C07259=1050.815,63.161,-79.530,170.792,33.398,156.273
C07260=1050.821,63.411,-79.547,170.794,33.400,156.273
C07261=1050.828,63.661,-79.565,170.795,33.402,156.273
C07262=1050.834,63.909,-79.583,170.797,33.404,156.274
C07263=1050.840,64.158,-79.601,170.799,33.406,156.274
C07264=1050.846,64.408,-79.619,170.800,33.407,156.274
C07265=1050.853,64.657,-79.636,170.802,33.410,156.275
C07266=1050.859,64.907,-79.654,170.804,33.412,156.275
C07267=1050.864,65.156,-79.671,170.805,33.414,156.276
C07268=1050.871,65.405,-79.689,170.807,33.416,156.276
C07269=1050.877,65.655,-79.707,170.809,33.418,156.276
C07270=1050.883,65.903,-79.725,170.810,33.420,156.276
C07271=1050.890,66.153,-79.742,170.812,33.422,156.277
C07272=1050.896,66.402,-79.760,170.813,33.424,156.277
C07273=1050.902,66.652,-79.778,170.815,33.426,156.277
C07274=1050.908,66.901,-79.795,170.817,33.428,156.278
C07275=1050.915,67.151,-79.813,170.818,33.430,156.278
C07276=1050.920,67.399,-79.831,170.820,33.432,156.278
C07277=1050.926,67.649,-79.849,170.822,33.434,156.279
C07278=1050.933,67.898,-79.867,170.823,33.436,156.279
C07279=1050.939,68.147,-79.884,170.825,33.438,156.279
C07280=1050.945,68.396,-79.903,170.826,33.440,156.280
C07281=1050.951,68.646,-79.921,170.828,33.442,156.280
C07282=1050.958,68.895,-79.938,170.830,33.444,156.280
C07283=1050.964,69.145,-79.956,170.831,33.446,156.281
C07284=1050.970,69.394,-79.974,170.833,33.449,156.281
C07285=1050.976,69.643,-79.992,170.835,33.451,156.281
C07286=1050.982,69.893,-80.010,170.836,33.453,156.282
C07287=1050.989,70.142,-80.027,170.838,33.455,156.282
C07288=1050.995,70.390,-80.045,170.839,33.457,156.282
C07289=1051.001,70.640,-80.063,170.841,33.459,156.283
C07290=1051.007,70.890,-80.081,170.843,33.461,156.283
C07291=1051.013,71.138,-80.099,170.844,33.463,156.283
C07292=1051.019,71.388,-80.117,170.846,33.465,156.284
C07293=1051.025,71.638,-80.135,170.847,33.467,156.284
C07294=1051.031,71.887,-80.154,170.849,33.469,156.284
C07295=1051.037,72.136,-80.172,170.851,33.471,156.285
C07296=1051.044,72.385,-80.190,170.852,33.473,156.285
C07297=1051.050,72.635,-80.208,170.854,33.475,156.285
C07298=1051.056,72.884,-80.225,170.856,33.478,156.286
C07299=1051.062,73.133,-80.244,170.857,33.479,156.286
C07300=1051.068,73.382,-80.262,170.859,33.481,156.286
C07301=1051.075,73.632,-80.280,170.861,33.483,156.287
C07302=1051.080,73.881,-80.298,170.863,33.485,156.287
C07303=1051.086,74.130,-80.316,170.865,33.487,156.287
C07304=1051.093,74.379,-80.335,170.866,33.490,156.288
C07305=1051.099,74.629,-80.352,170.868,33.492,156.288
C07306=1051.105,74.878,-80.371,170.870,33.494,156.288
C07307=1051.111,75.127,-80.389,170.871,33.496,156.289
C07308=1051.117,75.376,-80.407,170.873,33.498,156.289
C07309=1051.124,75.626,-80.425,170.874,33.500,156.289
C07310=1051.130,75.874,-80.443,170.876,33.502,156.290
C07311=1051.136,76.124,-80.461,170.878,33.504,156.290
C07312=1051.142,76.373,-80.480,170.879,33.506,156.291
C07313=1051.148,76.623,-80.497,170.881,33.508,156.291
C07314=1051.154,76.871,-80.516,170.883,33.510,156.291
C07315=1051.160,77.121,-80.534,170.884,33.512,156.291
C07316=1051.167,77.407,-80.555,170.886,33.515,156.292
C07317=1051.175,77.693,-80.576,170.888,33.517,156.292
C07318=1051.182,77.978,-80.597,170.890,33.519,156.293
C07319=1051.189,78.264,-80.618,170.892,33.522,156.293
C07320=1051.195,78.513,-80.636,170.893,33.524,156.293
C07321=1051.201,78.762,-80.654,170.895,33.526,156.294
C07322=1051.207,79.011,-80.673,170.897,33.528,156.294
C07323=1051.213,79.261,-80.691,170.898,33.530,156.294
C07324=1051.219,79.510,-80.710,170.900,33.532,156.295
C07325=1051.225,79.759,-80.729,170.901,33.534,156.295
C07326=1051.231,80.009,-80.746,170.903,33.536,156.295
C07327=1051.237,80.257,-80.765,170.905,33.538,156.296
C07328=1051.244,80.506,-80.783,170.906,33.541,156.296
C07329=1051.250,80.756,-80.801,170.908,33.543,156.297
C07330=1051.255,81.006,-80.821,170.909,33.545,156.297
C07331=1051.262,81.255,-80.839,170.911,33.547,156.297
C07332=1051.267,81.504,-80.857,170.913,33.549,156.298
C07333=1051.274,81.753,-80.875,170.914,33.551,156.298
C07334=1051.280,82.002,-80.894,170.916,33.553,156.298
C07335=1051.286,82.252,-80.913,170.918,33.555,156.299
C07336=1051.292,82.501,-80.931,170.919,33.558,156.299
C07337=1051.298,82.750,-80.950,170.921,33.560,156.299
C07338=1051.304,82.999,-80.968,170.922,33.562,156.300
C07339=1051.310,83.249,-80.986,170.924,33.564,156.300
C07340=1051.316,83.498,-81.005,170.926,33.566,156.300
C07341=1051.322,83.747,-81.024,170.927,33.568,156.301
C07342=1051.329,83.996,-81.043,170.929,33.570,156.301
C07343=1051.335,84.246,-81.061,170.931,33.572,156.301
C07344=1051.340,84.495,-81.080,170.933,33.574,156.302
C07345=1051.347,84.744,-81.098,170.935,33.576,156.302
C07346=1051.353,84.993,-81.117,170.936,33.579,156.302
C07347=1051.359,85.242,-81.135,170.938,33.580,156.303
C07348=1051.365,85.492,-81.153,170.940,33.582,156.303
C07349=1051.371,85.741,-81.173,170.941,33.584,156.303
C07350=1051.378,85.990,-81.191,170.943,33.586,156.304
C07351=1051.384,86.239,-81.210,170.945,33.589,156.304
C07352=1051.390,86.489,-81.229,170.946,33.591,156.304
C07353=1051.396,86.738,-81.248,170.948,33.593,156.305
C07354=1051.402,86.987,-81.265,170.949,33.595,156.305
C07355=1051.408,87.236,-81.284,170.951,33.597,156.305
C07356=1051.415,87.485,-81.303,170.953,33.599,156.306
C07357=1051.420,87.735,-81.322,170.954,33.601,156.306
C07358=1051.427,87.984,-81.341,170.956,33.603,156.307
C07359=1051.433,88.233,-81.359,170.958,33.605,156.307
C07360=1051.439,88.482,-81.378,170.959,33.607,156.307
C07361=1051.445,88.732,-81.397,170.961,33.609,156.307
C07362=1051.452,88.981,-81.416,170.963,33.612,156.308
C07363=1051.458,89.230,-81.434,170.964,33.614,156.308
C07364=1051.464,89.480,-81.452,170.966,33.616,156.309
C07365=1051.470,89.729,-81.472,170.968,33.618,156.309
C07366=1051.476,89.978,-81.490,170.969,33.620,156.309
C07367=1051.483,90.227,-81.509,170.971,33.622,156.310
C07368=1051.489,90.476,-81.528,170.972,33.624,156.310
C07369=1051.495,90.726,-81.547,170.974,33.626,156.310
C07370=1051.501,90.975,-81.565,170.976,33.628,156.311
C07371=1051.507,91.224,-81.585,170.977,33.631,156.311
C07372=1051.513,91.473,-81.603,170.979,33.633,156.311
C07373=1051.519,91.723,-81.623,170.981,33.634,156.312
C07374=1051.525,91.972,-81.641,170.982,33.636,156.312
C07375=1051.531,92.221,-81.660,170.984,33.639,156.312
C07376=1051.537,92.469,-81.679,170.985,33.641,156.313
C07377=1051.543,92.719,-81.699,170.988,33.643,156.313
C07378=1051.549,92.968,-81.717,170.990,33.645,156.314
C07379=1051.555,93.217,-81.737,170.991,33.647,156.314
C07380=1051.562,93.504,-81.758,170.993,33.650,156.314
C07381=1051.569,93.789,-81.780,170.995,33.652,156.315
C07382=1051.576,94.075,-81.802,170.997,33.655,156.315
C07383=1051.583,94.360,-81.824,170.999,33.657,156.315
C07384=1051.589,94.609,-81.842,171.000,33.659,156.316
C07385=1051.595,94.858,-81.862,171.002,33.662,156.316
C07386=1051.602,95.107,-81.881,171.004,33.664,156.317
C07387=1051.608,95.356,-81.900,171.005,33.666,156.317
C07388=1051.613,95.606,-81.920,171.007,33.667,156.317
C07389=1051.620,95.855,-81.938,171.009,33.670,156.318
C07390=1051.625,96.104,-81.957,171.010,33.672,156.318
C07391=1051.632,96.353,-81.976,171.012,33.674,156.318
C07392=1051.638,96.602,-81.996,171.014,33.676,156.319
C07393=1051.644,96.851,-82.015,171.015,33.678,156.319
C07394=1051.650,97.101,-82.034,171.017,33.680,156.319
C07395=1051.656,97.350,-82.053,171.019,33.682,156.320
C07396=1051.662,97.599,-82.072,171.020,33.684,156.320
C07397=1051.669,97.848,-82.091,171.022,33.687,156.320
C07398=1051.674,98.097,-82.110,171.024,33.689,156.321
C07399=1051.680,98.347,-82.130,171.025,33.691,156.321
C07400=1051.687,98.597,-82.149,171.027,33.693,156.321
C07401=1051.693,98.845,-82.169,171.028,33.695,156.322
C07402=1051.700,99.094,-82.187,171.030,33.697,156.322
C07403=1051.705,99.344,-82.207,171.032,33.699,156.323
C07404=1051.712,99.592,-82.226,171.033,33.701,156.323
C07405=1051.718,99.842,-82.245,171.036,33.704,156.323
C07406=1051.724,100.091,-82.264,171.038,33.706,156.324
C07407=1051.730,100.340,-82.283,171.039,33.708,156.324
C07408=1051.736,100.589,-82.303,171.041,33.710,156.324
C07409=1051.742,100.838,-82.322,171.043,33.712,156.325
C07410=1051.748,101.088,-82.341,171.044,33.714,156.325
C07411=1051.754,101.337,-82.361,171.046,33.716,156.325
C07412=1051.760,101.587,-82.380,171.048,33.719,156.326
C07413=1051.767,101.835,-82.400,171.049,33.721,156.326
C07414=1051.773,102.085,-82.419,171.051,33.723,156.326
C07415=1051.778,102.334,-82.438,171.053,33.725,156.327
C07416=1051.784,102.583,-82.458,171.054,33.727,156.327
C07417=1051.790,102.832,-82.478,171.056,33.729,156.328
C07418=1051.797,103.081,-82.497,171.058,33.732,156.328
C07419=1051.802,103.330,-82.516,171.059,33.733,156.328
C07420=1051.808,103.579,-82.536,171.061,33.735,156.329
C07421=1051.814,103.829,-82.555,171.062,33.738,156.329
C07422=1051.821,104.078,-82.576,171.064,33.740,156.329
C07423=1051.826,104.327,-82.595,171.066,33.742,156.330
C07424=1051.833,104.576,-82.614,171.067,33.744,156.330
C07425=1051.839,104.825,-82.633,171.069,33.746,156.330
C07426=1051.845,105.074,-82.653,171.071,33.748,156.331
C07427=1051.850,105.324,-82.673,171.072,33.751,156.331
C07428=1051.856,105.572,-82.693,171.074,33.753,156.332
C07429=1051.863,105.822,-82.711,171.076,33.755,156.332
C07430=1051.869,106.071,-82.732,171.078,33.757,156.332
C07431=1051.875,106.321,-82.751,171.080,33.759,156.333
C07432=1051.881,106.569,-82.771,171.082,33.761,156.333
C07433=1051.887,106.819,-82.790,171.083,33.764,156.333
C07434=1051.893,107.068,-82.810,171.085,33.766,156.334
C07435=1051.899,107.317,-82.829,171.087,33.768,156.334
C07436=1051.906,107.566,-82.849,171.088,33.770,156.335
C07437=1051.912,107.815,-82.869,171.090,33.772,156.335
C07438=1051.918,108.064,-82.888,171.092,33.774,156.335
C07439=1051.924,108.313,-82.908,171.093,33.777,156.336
C07440=1051.929,108.563,-82.927,171.095,33.779,156.336
C07441=1051.936,108.812,-82.948,171.097,33.781,156.336
C07442=1051.943,109.061,-82.967,171.098,33.783,156.337
C07443=1051.948,109.310,-82.986,171.100,33.785,156.337
C07444=1051.955,109.596,-83.009,171.102,33.788,156.337
C07445=1051.963,109.881,-83.032,171.104,33.790,156.338
C07446=1051.970,110.166,-83.054,171.106,33.792,156.338
C07447=1051.976,110.452,-83.077,171.108,33.795,156.339
C07448=1051.982,110.701,-83.097,171.110,33.797,156.339
C07449=1051.988,110.951,-83.117,171.111,33.799,156.339
C07450=1051.994,111.200,-83.137,171.113,33.801,156.340
C07451=1052.000,111.449,-83.157,171.115,33.803,156.340
C07452=1052.006,111.698,-83.176,171.117,33.806,156.341
C07453=1052.012,111.947,-83.196,171.119,33.808,156.341
C07454=1052.019,112.197,-83.216,171.121,33.810,156.341
C07455=1052.025,112.445,-83.236,171.122,33.812,156.342
C07456=1052.030,112.695,-83.255,171.124,33.814,156.342
C07457=1052.036,112.944,-83.275,171.126,33.816,156.342
C07458=1052.043,113.193,-83.296,171.127,33.819,156.343
C07459=1052.049,113.442,-83.316,171.129,33.821,156.343
C07460=1052.055,113.691,-83.335,171.131,33.823,156.343
C07461=1052.061,113.940,-83.355,171.132,33.825,156.344
C07462=1052.067,114.190,-83.375,171.134,33.827,156.344
C07463=1052.073,114.439,-83.395,171.136,33.830,156.345
C07464=1052.079,114.688,-83.416,171.137,33.831,156.345
C07465=1052.085,114.936,-83.436,171.139,33.834,156.345
C07466=1052.091,115.186,-83.456,171.141,33.836,156.346
C07467=1052.097,115.435,-83.475,171.142,33.838,156.346
C07468=1052.102,115.685,-83.496,171.144,33.840,156.346
C07469=1052.108,115.933,-83.516,171.146,33.843,156.347
C07470=1052.115,116.183,-83.536,171.147,33.845,156.347
C07471=1052.121,116.432,-83.556,171.149,33.847,156.348
C07472=1052.126,116.681,-83.577,171.152,33.849,156.348
C07473=1052.132,116.930,-83.597,171.154,33.852,156.348
C07474=1052.139,117.179,-83.617,171.155,33.854,156.349
C07475=1052.144,117.428,-83.637,171.157,33.856,156.349
C07476=1052.150,117.677,-83.657,171.159,33.858,156.349
C07477=1052.156,117.926,-83.677,171.160,33.860,156.350
C07478=1052.162,118.175,-83.698,171.162,33.863,156.350
C07479=1052.168,118.424,-83.718,171.164,33.865,156.351
C07480=1052.174,118.673,-83.738,171.165,33.867,156.351
C07481=1052.180,118.923,-83.759,171.167,33.869,156.351
C07482=1052.186,119.172,-83.779,171.169,33.872,156.352
C07483=1052.191,119.421,-83.799,171.170,33.874,156.352
C07484=1052.197,119.670,-83.819,171.172,33.876,156.352
C07485=1052.204,119.919,-83.839,171.174,33.878,156.353
C07486=1052.210,120.168,-83.859,171.176,33.880,156.353
C07487=1052.215,120.417,-83.880,171.177,33.883,156.354
C07488=1052.222,120.667,-83.900,171.179,33.885,156.354
C07489=1052.228,120.915,-83.920,171.181,33.887,156.354
C07490=1052.233,121.165,-83.941,171.182,33.889,156.355
C07491=1052.240,121.414,-83.961,171.185,33.892,156.355
C07492=1052.246,121.663,-83.981,171.187,33.894,156.356
C07493=1052.252,121.912,-84.003,171.188,33.896,156.356
C07494=1052.258,122.161,-84.023,171.190,33.898,156.356
C07495=1052.264,122.410,-84.043,171.192,33.900,156.357
C07496=1052.270,122.659,-84.063,171.194,33.903,156.357
C07497=1052.276,122.908,-84.083,171.195,33.905,156.357
C07498=1052.282,123.157,-84.103,171.197,33.907,156.358
C07499=1052.288,123.407,-84.124,171.199,33.909,156.358
C07500=1052.294,123.656,-84.144,171.200,33.911,156.358
C07501=1052.300,123.905,-84.165,171.202,33.914,156.359
C07502=1052.306,124.153,-84.185,171.204,33.916,156.359
C07503=1052.312,124.403,-84.206,171.206,33.918,156.360
C07504=1052.318,124.652,-84.226,171.207,33.920,156.360
C07505=1052.324,124.901,-84.246,171.209,33.922,156.360
C07506=1052.330,125.150,-84.268,171.211,33.925,156.361
C07507=1052.336,125.399,-84.288,171.213,33.926,156.361
C07508=1052.343,125.684,-84.311,171.215,33.929,156.362
C07509=1052.350,125.970,-84.334,171.218,33.932,156.362
C07510=1052.357,126.256,-84.358,171.220,33.934,156.362
C07511=1052.364,126.541,-84.382,171.222,33.937,156.363
C07512=1052.370,126.790,-84.402,171.223,33.939,156.363
C07513=1052.377,127.039,-84.423,171.225,33.941,156.364
C07514=1052.382,127.288,-84.443,171.227,33.943,156.364
C07515=1052.389,127.537,-84.463,171.229,33.945,156.364
C07516=1052.394,127.786,-84.485,171.230,33.948,156.365
C07517=1052.401,128.036,-84.505,171.232,33.950,156.365
C07518=1052.407,128.284,-84.525,171.234,33.952,156.366
C07519=1052.413,128.534,-84.546,171.236,33.954,156.366
C07520=1052.419,128.782,-84.567,171.237,33.956,156.366
C07521=1052.426,129.032,-84.587,171.239,33.958,156.367
C07522=1052.431,129.281,-84.608,171.241,33.960,156.367
C07523=1052.438,129.530,-84.629,171.243,33.963,156.367
C07524=1052.444,129.779,-84.648,171.244,33.965,156.368
C07525=1052.450,130.028,-84.670,171.246,33.967,156.368
C07526=1052.456,130.277,-84.690,171.249,33.969,156.369
C07527=1052.462,130.527,-84.711,171.251,33.971,156.369
C07528=1052.468,130.775,-84.732,171.252,33.973,156.369
C07529=1052.475,131.024,-84.752,171.254,33.976,156.370
C07530=1052.481,131.273,-84.774,171.256,33.978,156.370
C07531=1052.487,131.522,-84.794,171.258,33.980,156.370
C07532=1052.493,131.772,-84.815,171.259,33.982,156.371
C07533=1052.499,132.020,-84.835,171.261,33.985,156.371
C07534=1052.505,132.270,-84.856,171.263,33.987,156.371
C07535=1052.511,132.519,-84.877,171.265,33.989,156.372
C07536=1052.517,132.768,-84.898,171.266,33.991,156.372
C07537=1052.523,133.017,-84.919,171.268,33.994,156.373
C07538=1052.529,133.266,-84.940,171.270,33.996,156.373
C07539=1052.535,133.515,-84.961,171.272,33.998,156.373
C07540=1052.541,133.764,-84.982,171.273,34.000,156.374
C07541=1052.546,134.013,-85.003,171.275,34.003,156.374
C07542=1052.553,134.262,-85.024,171.278,34.005,156.375
C07543=1052.559,134.511,-85.044,171.280,34.007,156.375
C07544=1052.565,134.760,-85.066,171.282,34.009,156.375
C07545=1052.571,135.009,-85.086,171.283,34.012,156.376
C07546=1052.577,135.258,-85.108,171.285,34.014,156.376
C07547=1052.582,135.507,-85.129,171.287,34.016,156.377
C07548=1052.589,135.756,-85.149,171.289,34.018,156.377
C07549=1052.595,136.005,-85.171,171.290,34.021,156.377
C07550=1052.600,136.255,-85.191,171.292,34.022,156.378
C07551=1052.607,136.503,-85.212,171.294,34.025,156.378
C07552=1052.613,136.752,-85.234,171.296,34.027,156.378
C07553=1052.619,137.002,-85.255,171.298,34.030,156.379
C07554=1052.625,137.250,-85.275,171.299,34.031,156.379
C07555=1052.631,137.499,-85.297,171.301,34.034,156.380
C07556=1052.637,137.749,-85.318,171.303,34.036,156.380
C07557=1052.643,137.998,-85.339,171.306,34.038,156.380
C07558=1052.650,138.246,-85.360,171.307,34.041,156.381
C07559=1052.655,138.496,-85.381,171.309,34.043,156.381
C07560=1052.661,138.745,-85.402,171.311,34.045,156.382
C07561=1052.667,138.994,-85.424,171.313,34.047,156.382
C07562=1052.673,139.242,-85.445,171.315,34.050,156.382
C07563=1052.679,139.492,-85.466,171.316,34.052,156.383
C07564=1052.685,139.741,-85.487,171.318,34.054,156.383
C07565=1052.691,139.990,-85.508,171.320,34.056,156.384
C07566=1052.697,140.239,-85.530,171.322,34.059,156.384
C07567=1052.702,140.488,-85.551,171.324,34.061,156.384
C07568=1052.709,140.737,-85.572,171.325,34.063,156.385
C07569=1052.715,140.986,-85.593,171.327,34.066,156.385
C07570=1052.721,141.235,-85.615,171.329,34.068,156.386
C07571=1052.727,141.484,-85.636,171.332,34.070,156.386
C07572=1052.733,141.770,-85.660,171.334,34.073,156.386
C07573=1052.741,142.054,-85.685,171.336,34.075,156.387
C07574=1052.747,142.339,-85.710,171.338,34.078,156.387
C07575=1052.754,142.625,-85.734,171.340,34.081,156.388
C07576=1052.760,142.874,-85.756,171.342,34.083,156.388
C07577=1052.767,143.123,-85.777,171.344,34.086,156.389
C07578=1052.772,143.372,-85.798,171.345,34.088,156.389
C07579=1052.778,143.621,-85.820,171.347,34.090,156.389
C07580=1052.785,143.870,-85.841,171.349,34.092,156.390
C07581=1052.790,144.119,-85.863,171.351,34.095,156.390
C07582=1052.796,144.368,-85.884,171.353,34.097,156.391
C07583=1052.802,144.617,-85.906,171.355,34.099,156.391
C07584=1052.808,144.866,-85.926,171.357,34.102,156.391
C07585=1052.814,145.115,-85.948,171.359,34.103,156.392
C07586=1052.820,145.365,-85.970,171.361,34.106,156.392
C07587=1052.826,145.614,-85.991,171.363,34.108,156.393
C07588=1052.832,145.862,-86.013,171.365,34.111,156.393
C07589=1052.838,146.111,-86.034,171.367,34.113,156.393
C07590=1052.844,146.361,-86.056,171.368,34.115,156.394
C07591=1052.850,146.609,-86.077,171.370,34.117,156.394
C07592=1052.856,146.858,-86.099,171.372,34.119,156.395
C07593=1052.862,147.108,-86.120,171.374,34.122,156.395
C07594=1052.868,147.357,-86.142,171.376,34.124,156.395
C07595=1052.874,147.605,-86.164,171.378,34.126,156.396
C07596=1052.880,147.854,-86.186,171.379,34.129,156.396
C07597=1052.886,148.103,-86.207,171.381,34.131,156.397
C07598=1052.892,148.352,-86.229,171.384,34.133,156.397
C07599=1052.898,148.601,-86.250,171.386,34.136,156.397
C07600=1052.904,148.850,-86.272,171.388,34.138,156.398
C07601=1052.910,149.099,-86.293,171.390,34.140,156.398
C07602=1052.917,149.348,-86.315,171.391,34.143,156.399
C07603=1052.922,149.597,-86.336,171.393,34.145,156.399
C07604=1052.928,149.846,-86.359,171.395,34.147,156.399
C07605=1052.934,150.095,-86.381,171.397,34.150,156.400
C07606=1052.940,150.344,-86.403,171.399,34.152,156.400
C07607=1052.946,150.593,-86.424,171.401,34.154,156.401
C07608=1052.952,150.842,-86.445,171.403,34.157,156.401
C07609=1052.958,151.090,-86.468,171.404,34.159,156.401
C07610=1052.964,151.340,-86.490,171.407,34.161,156.402
C07611=1052.970,151.589,-86.512,171.409,34.164,156.402
C07612=1052.975,151.838,-86.533,171.411,34.166,156.403
C07613=1052.982,152.086,-86.555,171.413,34.168,156.403
C07614=1052.988,152.336,-86.577,171.415,34.171,156.404
C07615=1052.994,152.585,-86.599,171.417,34.173,156.404
C07616=1053.000,152.834,-86.621,171.418,34.175,156.404
C07617=1053.006,153.082,-86.643,171.420,34.178,156.405
C07618=1053.012,153.331,-86.664,171.422,34.180,156.405
C07619=1053.018,153.581,-86.686,171.424,34.182,156.406
C07620=1053.023,153.830,-86.708,171.426,34.185,156.406
C07621=1053.030,154.079,-86.731,171.428,34.187,156.406
C07622=1053.036,154.328,-86.752,171.431,34.189,156.407
C07623=1053.042,154.576,-86.774,171.433,34.192,156.407
C07624=1053.047,154.825,-86.796,171.434,34.194,156.408
C07625=1053.053,155.074,-86.818,171.436,34.196,156.408
C07626=1053.060,155.323,-86.840,171.438,34.199,156.409
C07627=1053.065,155.573,-86.863,171.440,34.201,156.409
C07628=1053.071,155.822,-86.884,171.442,34.203,156.409
C07629=1053.077,156.070,-86.906,171.444,34.206,156.410
C07630=1053.083,156.319,-86.929,171.446,34.208,156.410
C07631=1053.089,156.568,-86.951,171.448,34.211,156.411
C07632=1053.095,156.817,-86.973,171.450,34.213,156.411
C07633=1053.101,157.066,-86.995,171.451,34.215,156.411
C07634=1053.107,157.315,-87.017,171.454,34.218,156.412
C07635=1053.113,157.564,-87.039,171.456,34.220,156.412
C07636=1053.120,157.849,-87.064,171.458,34.223,156.413
C07637=1053.127,158.134,-87.089,171.461,34.225,156.413
C07638=1053.134,158.418,-87.115,171.463,34.228,156.414
C07639=1053.141,158.704,-87.140,171.465,34.231,156.414
C07640=1053.146,158.952,-87.163,171.467,34.233,156.415
C07641=1053.152,159.201,-87.185,171.469,34.236,156.415
C07642=1053.158,159.450,-87.208,171.471,34.238,156.415
C07643=1053.164,159.700,-87.229,171.473,34.241,156.416
C07644=1053.171,159.948,-87.252,171.475,34.243,156.416
C07645=1053.176,160.198,-87.274,171.477,34.245,156.417
C07646=1053.183,160.446,-87.296,171.479,34.248,156.417
C07647=1053.189,160.695,-87.318,171.481,34.250,156.417
C07648=1053.194,160.944,-87.341,171.483,34.252,156.418
C07649=1053.200,161.193,-87.364,171.485,34.255,156.418
C07650=1053.206,161.443,-87.386,171.487,34.257,156.419
C07651=1053.212,161.691,-87.408,171.489,34.260,156.419
C07652=1053.217,161.940,-87.431,171.491,34.262,156.420
C07653=1053.223,162.189,-87.453,171.493,34.265,156.420
C07654=1053.228,162.438,-87.476,171.495,34.267,156.421
C07655=1053.235,162.687,-87.498,171.498,34.270,156.421
C07656=1053.241,162.935,-87.521,171.499,34.272,156.422
C07657=1053.246,163.185,-87.544,171.501,34.275,156.422
C07658=1053.252,163.434,-87.566,171.503,34.277,156.422
C07659=1053.258,163.682,-87.589,171.505,34.280,156.423
C07660=1053.264,163.931,-87.612,171.507,34.282,156.423
C07661=1053.269,164.181,-87.634,171.509,34.285,156.424
C07662=1053.274,164.429,-87.657,171.511,34.287,156.424
C07663=1053.281,164.678,-87.679,171.513,34.289,156.425
C07664=1053.287,164.927,-87.702,171.515,34.292,156.425
C07665=1053.292,165.175,-87.725,171.517,34.294,156.425
C07666=1053.298,165.425,-87.747,171.520,34.297,156.426
C07667=1053.304,165.674,-87.769,171.522,34.299,156.426
C07668=1053.310,165.922,-87.792,171.524,34.302,156.427
C07669=1053.316,166.171,-87.815,171.525,34.304,156.427
C07670=1053.321,166.420,-87.838,171.527,34.307,156.428
C07671=1053.327,166.669,-87.861,171.529,34.309,156.428
C07672=1053.334,166.918,-87.884,171.531,34.312,156.429
C07673=1053.339,167.167,-87.906,171.533,34.315,156.429
C07674=1053.345,167.416,-87.929,171.535,34.317,156.430
C07675=1053.351,167.665,-87.952,171.538,34.320,156.430
C07676=1053.357,167.914,-87.974,171.540,34.322,156.430
C07677=1053.363,168.162,-87.997,171.542,34.324,156.431
C07678=1053.368,168.411,-88.020,171.544,34.327,156.431
C07679=1053.374,168.660,-88.043,171.546,34.329,156.432
C07680=1053.380,168.909,-88.066,171.548,34.332,156.432
C07681=1053.386,169.158,-88.089,171.550,34.334,156.433
C07682=1053.392,169.407,-88.111,171.552,34.337,156.433
C07683=1053.398,169.656,-88.134,171.554,34.339,156.433
C07684=1053.404,169.904,-88.157,171.556,34.342,156.434
C07685=1053.409,170.153,-88.180,171.559,34.344,156.434
C07686=1053.415,170.402,-88.203,171.561,34.347,156.435
C07687=1053.422,170.651,-88.225,171.563,34.349,156.435
C07688=1053.428,170.900,-88.249,171.565,34.352,156.436
C07689=1053.434,171.149,-88.271,171.567,34.354,156.436
C07690=1053.439,171.398,-88.294,171.569,34.357,156.437
C07691=1053.445,171.647,-88.317,171.571,34.359,156.437
C07692=1053.451,171.896,-88.340,171.573,34.362,156.438
C07693=1053.457,172.145,-88.363,171.575,34.364,156.438
C07694=1053.463,172.393,-88.386,171.577,34.366,156.438
C07695=1053.469,172.642,-88.409,171.580,34.369,156.439
C07696=1053.474,172.891,-88.432,171.582,34.371,156.439
C07697=1053.481,173.141,-88.455,171.584,34.374,156.440
C07698=1053.487,173.389,-88.478,171.586,34.376,156.440
C07699=1053.493,173.638,-88.501,171.588,34.379,156.441
C07700=1053.499,173.923,-88.527,171.590,34.382,156.441
C07701=1053.507,174.206,-88.554,171.592,34.384,156.442
C07702=1053.513,174.492,-88.580,171.595,34.388,156.442
C07703=1053.520,174.776,-88.606,171.597,34.390,156.443
C07704=1053.526,175.025,-88.629,171.600,34.393,156.443
C07705=1053.532,175.273,-88.652,171.602,34.395,156.444
C07706=1053.538,175.522,-88.675,171.604,34.398,156.444
C07707=1053.544,175.772,-88.699,171.606,34.400,156.444
C07708=1053.550,176.021,-88.722,171.608,34.403,156.445
C07709=1053.557,176.269,-88.745,171.610,34.405,156.445
C07710=1053.562,176.518,-88.768,171.612,34.408,156.446
C07711=1053.568,176.767,-88.791,171.614,34.410,156.446
C07712=1053.574,177.016,-88.814,171.616,34.413,156.447
C07713=1053.580,177.264,-88.838,171.620,34.415,156.447
C07714=1053.586,177.513,-88.861,171.622,34.418,156.448
C07715=1053.592,177.762,-88.883,171.624,34.420,156.448
C07716=1053.599,178.011,-88.907,171.626,34.423,156.449
C07717=1053.605,178.260,-88.930,171.628,34.425,156.449
C07718=1053.611,178.509,-88.953,171.630,34.427,156.449
C07719=1053.617,178.757,-88.976,171.632,34.430,156.450
C07720=1053.623,179.007,-89.000,171.634,34.432,156.450
C07721=1053.629,179.255,-89.023,171.636,34.435,156.451
C07722=1053.635,179.504,-89.046,171.639,34.437,156.451
C07723=1053.641,179.753,-89.069,171.641,34.440,156.452
C07724=1053.647,180.002,-89.093,171.643,34.442,156.452
C07725=1053.653,180.251,-89.116,171.645,34.445,156.453
C07726=1053.659,180.499,-89.139,171.647,34.447,156.453
C07727=1053.665,180.748,-89.163,171.650,34.450,156.453
C07728=1053.672,180.997,-89.186,171.652,34.452,156.454
C07729=1053.678,181.246,-89.209,171.654,34.455,156.454
C07730=1053.684,181.495,-89.233,171.656,34.457,156.455
C07731=1053.690,181.744,-89.256,171.659,34.460,156.455
C07732=1053.696,181.992,-89.279,171.661,34.462,156.456
C07733=1053.702,182.242,-89.303,171.663,34.465,156.456
C07734=1053.708,182.490,-89.326,171.665,34.468,156.457
C07735=1053.714,182.739,-89.349,171.667,34.470,156.457
C07736=1053.721,182.988,-89.373,171.669,34.473,156.458
C07737=1053.726,183.237,-89.396,171.672,34.475,156.458
C07738=1053.733,183.486,-89.420,171.674,34.478,156.458
C07739=1053.739,183.735,-89.443,171.677,34.480,156.459
C07740=1053.745,183.983,-89.467,171.679,34.483,156.459
C07741=1053.751,184.232,-89.490,171.681,34.485,156.460
C07742=1053.757,184.481,-89.514,171.683,34.488,156.460
C07743=1053.762,184.729,-89.538,171.685,34.490,156.461
C07744=1053.769,184.979,-89.561,171.687,34.493,156.461
C07745=1053.775,185.227,-89.585,171.689,34.496,156.462
C07746=1053.780,185.476,-89.609,171.691,34.498,156.462
C07747=1053.786,185.725,-89.632,171.695,34.501,156.463
C07748=1053.792,185.974,-89.657,171.697,34.504,156.463
C07749=1053.798,186.222,-89.680,171.699,34.506,156.464
C07750=1053.803,186.471,-89.705,171.701,34.509,156.464
C07751=1053.809,186.720,-89.728,171.703,34.512,156.465
C07752=1053.815,186.969,-89.752,171.705,34.514,156.465
C07753=1053.821,187.217,-89.776,171.707,34.517,156.466
C07754=1053.827,187.466,-89.800,171.709,34.519,156.466
C07755=1053.832,187.715,-89.823,171.712,34.523,156.467
C07756=1053.838,187.964,-89.847,171.715,34.525,156.467
C07757=1053.844,188.213,-89.872,171.717,34.528,156.468
C07758=1053.850,188.461,-89.895,171.719,34.531,156.468
C07759=1053.856,188.710,-89.920,171.721,34.533,156.469
C07760=1053.862,188.959,-89.943,171.723,34.536,156.469
C07761=1053.867,189.208,-89.967,171.725,34.538,156.470
C07762=1053.873,189.456,-89.991,171.728,34.541,156.470
C07763=1053.879,189.706,-90.016,171.730,34.544,156.471
C07764=1053.886,189.990,-90.043,171.733,34.547,156.471
C07765=1053.892,190.273,-90.070,171.735,34.550,156.472
C07766=1053.900,190.558,-90.098,171.738,34.553,156.472
C07767=1053.906,190.842,-90.125,171.740,34.556,156.473
C07768=1053.912,191.090,-90.149,171.742,34.559,156.473
C07769=1053.918,191.339,-90.174,171.746,34.561,156.474
C07770=1053.924,191.587,-90.197,171.748,34.564,156.474
C07771=1053.930,191.837,-90.221,171.750,34.567,156.475
C07772=1053.936,192.086,-90.245,171.752,34.569,156.475
C07773=1053.942,192.335,-90.269,171.754,34.573,156.476
C07774=1053.948,192.583,-90.293,171.756,34.575,156.476
C07775=1053.954,192.833,-90.318,171.759,34.578,156.477
C07776=1053.960,193.081,-90.341,171.761,34.581,156.477
C07777=1053.966,193.330,-90.366,171.764,34.583,156.478
C07778=1053.972,193.578,-90.390,171.766,34.586,156.478
C07779=1053.978,193.827,-90.415,171.768,34.589,156.479
C07780=1053.984,194.075,-90.439,171.770,34.591,156.479
C07781=1053.990,194.325,-90.463,171.773,34.594,156.480
C07782=1053.996,194.573,-90.487,171.775,34.597,156.480
C07783=1054.002,194.822,-90.512,171.777,34.599,156.481
C07784=1054.007,195.071,-90.536,171.780,34.602,156.481
C07785=1054.014,195.320,-90.560,171.782,34.605,156.482
C07786=1054.019,195.568,-90.584,171.785,34.608,156.482
C07787=1054.026,195.817,-90.608,171.787,34.610,156.483
C07788=1054.031,196.066,-90.632,171.789,34.613,156.483
C07789=1054.038,196.314,-90.657,171.791,34.616,156.484
C07790=1054.043,196.563,-90.681,171.793,34.618,156.484
C07791=1054.050,196.812,-90.705,171.797,34.621,156.485
C07792=1054.056,197.061,-90.730,171.799,34.624,156.485
C07793=1054.062,197.309,-90.754,171.801,34.627,156.486
C07794=1054.068,197.559,-90.778,171.803,34.629,156.486
C07795=1054.073,197.807,-90.803,171.806,34.632,156.487
C07796=1054.080,198.056,-90.827,171.808,34.635,156.487
C07797=1054.085,198.304,-90.852,171.810,34.637,156.488
C07798=1054.092,198.553,-90.876,171.813,34.640,156.488
C07799=1054.098,198.802,-90.901,171.815,34.643,156.489
C07800=1054.104,199.050,-90.925,171.818,34.646,156.489
C07801=1054.110,199.299,-90.949,171.820,34.649,156.490
C07802=1054.116,199.549,-90.974,171.822,34.651,156.490
C07803=1054.122,199.796,-90.998,171.824,34.654,156.491
C07804=1054.128,200.046,-91.023,171.827,34.657,156.491
C07805=1054.135,200.295,-91.047,171.830,34.659,156.492
C07806=1054.140,200.543,-91.072,171.832,34.662,156.492
C07807=1054.147,200.792,-91.096,171.835,34.665,156.493
C07808=1054.153,201.041,-91.120,171.837,34.667,156.493
C07809=1054.159,201.289,-91.145,171.839,34.670,156.494
C07810=1054.165,201.538,-91.169,171.841,34.673,156.494
C07811=1054.171,201.786,-91.195,171.845,34.676,156.495
C07812=1054.177,202.035,-91.219,171.847,34.678,156.495
C07813=1054.183,202.284,-91.244,171.849,34.682,156.496
C07814=1054.189,202.533,-91.268,171.851,34.684,156.496
C07815=1054.195,202.781,-91.293,171.854,34.687,156.497
C07816=1054.201,203.030,-91.318,171.856,34.690,156.498
C07817=1054.206,203.279,-91.342,171.858,34.693,156.498
C07818=1054.213,203.527,-91.368,171.861,34.696,156.499
C07819=1054.218,203.777,-91.392,171.864,34.698,156.499
C07820=1054.224,204.024,-91.417,171.866,34.701,156.500
C07821=1054.230,204.273,-91.443,171.868,34.705,156.500
C07822=1054.236,204.522,-91.467,171.870,34.707,156.501
C07823=1054.242,204.771,-91.493,171.873,34.710,156.501
C07824=1054.248,205.019,-91.516,171.876,34.713,156.502
C07825=1054.255,205.268,-91.542,171.878,34.716,156.502
C07826=1054.260,205.517,-91.566,171.881,34.719,156.503
C07827=1054.266,205.765,-91.591,171.883,34.721,156.503
C07828=1054.291,206.816,-91.697,172.092,34.813,156.518
C07829=1054.298,207.059,-91.722,172.094,34.817,156.519
C07830=1054.304,207.301,-91.748,172.096,34.821,156.520
C07831=1054.311,207.543,-91.772,172.098,34.824,156.520
C07832=1054.316,207.785,-91.797,172.100,34.828,156.521
C07833=1054.323,208.027,-91.823,172.101,34.832,156.522
C07834=1054.329,208.269,-91.848,172.104,34.835,156.523
C07835=1054.335,208.511,-91.873,172.106,34.839,156.523
C07836=1054.341,208.753,-91.898,172.107,34.842,156.524
C07837=1054.347,209.001,-91.924,172.109,34.846,156.525
C07838=1054.353,209.251,-91.951,172.112,34.850,156.525
C07839=1054.360,209.499,-91.977,172.114,34.853,156.526
C07840=1054.366,209.748,-92.002,172.115,34.857,156.527
C07841=1054.373,209.996,-92.028,172.117,34.861,156.528
C07842=1054.379,210.245,-92.055,172.120,34.864,156.528
C07843=1054.385,210.493,-92.081,172.122,34.868,156.529
C07844=1054.392,210.741,-92.107,172.123,34.872,156.530
C07845=1054.397,210.990,-92.133,172.125,34.876,156.530
C07846=1054.404,211.239,-92.159,172.128,34.879,156.531
C07847=1054.410,211.488,-92.186,172.130,34.883,156.532
C07848=1054.416,211.736,-92.211,172.131,34.886,156.533
C07849=1054.423,211.984,-92.237,172.133,34.890,156.533
C07850=1054.429,212.233,-92.264,172.136,34.894,156.534
C07851=1054.436,212.481,-92.290,172.138,34.897,156.535
C07852=1054.441,212.730,-92.316,172.139,34.901,156.535
C07853=1054.448,212.979,-92.342,172.141,34.905,156.536
C07854=1054.454,213.227,-92.369,172.143,34.908,156.537
C07855=1054.460,213.475,-92.395,172.146,34.912,156.538
C07856=1054.466,213.724,-92.421,172.147,34.916,156.538
C07857=1054.473,213.973,-92.447,172.149,34.920,156.539
C07858=1054.479,214.222,-92.474,172.152,34.923,156.540
C07859=1054.485,214.470,-92.500,172.154,34.927,156.541
C07860=1054.492,214.719,-92.527,172.155,34.930,156.541
C07861=1054.498,214.967,-92.553,172.157,34.934,156.542
C07862=1054.504,215.216,-92.579,172.160,34.938,156.543
C07863=1054.510,215.464,-92.605,172.162,34.941,156.543
C07864=1054.517,215.713,-92.632,172.164,34.945,156.544
C07865=1054.523,215.961,-92.658,172.165,34.949,156.545
C07866=1054.529,216.210,-92.685,172.168,34.952,156.546
C07867=1054.535,216.458,-92.712,172.170,34.956,156.546
C07868=1054.542,216.706,-92.738,172.172,34.959,156.547
C07869=1054.548,216.956,-92.764,172.174,34.963,156.548
C07870=1054.554,217.204,-92.790,172.176,34.967,156.549
C07871=1054.560,217.452,-92.817,172.178,34.971,156.549
C07872=1054.567,217.701,-92.843,172.180,34.975,156.550
C07873=1054.573,217.950,-92.870,172.182,34.978,156.551
C07874=1054.580,218.198,-92.897,172.185,34.982,156.551
C07875=1054.586,218.447,-92.923,172.186,34.985,156.552
C07876=1054.592,218.695,-92.950,172.188,34.989,156.553
C07877=1054.599,218.944,-92.976,172.190,34.993,156.554
C07878=1054.605,219.192,-93.003,172.193,34.996,156.554
C07879=1054.612,219.441,-93.029,172.195,34.999,156.555
C07880=1054.617,219.689,-93.056,172.197,35.003,156.556
C07881=1054.623,219.938,-93.083,172.198,35.006,156.556
C07882=1054.630,220.186,-93.109,172.201,35.010,156.557
C07883=1054.636,220.435,-93.136,172.203,35.014,156.558
C07884=1054.643,220.683,-93.162,172.205,35.017,156.559
C07885=1054.649,220.927,-93.189,172.207,35.021,156.559
C07886=1054.655,221.173,-93.215,172.210,35.025,156.560
C07887=1054.662,221.417,-93.241,172.211,35.028,156.561
C07888=1054.667,221.662,-93.268,172.213,35.032,156.561
C07889=1054.674,221.906,-93.294,172.215,35.035,156.562
C07890=1054.680,222.151,-93.321,172.218,35.039,156.563
C07891=1054.686,222.396,-93.347,172.220,35.043,156.564
C07892=1054.692,222.641,-93.374,172.222,35.046,156.564
C07893=1054.699,222.888,-93.400,172.223,35.050,156.565
C07894=1054.705,223.137,-93.427,172.226,35.053,156.566
C07895=1054.711,223.386,-93.454,172.228,35.057,156.566
C07896=1054.717,223.635,-93.481,172.230,35.061,156.567
C07897=1054.723,223.883,-93.508,172.233,35.064,156.568
C07898=1054.730,224.132,-93.536,172.235,35.068,156.569
C07899=1054.736,224.380,-93.562,172.237,35.072,156.569
C07900=1054.742,224.628,-93.588,172.238,35.075,156.570
C07901=1054.749,224.877,-93.616,172.241,35.079,156.571
C07902=1054.755,225.126,-93.643,172.243,35.082,156.571
C07903=1054.761,225.374,-93.670,172.245,35.086,156.572
C07904=1054.767,225.622,-93.697,172.247,35.090,156.573
C07905=1054.773,225.871,-93.724,172.250,35.093,156.574
C07906=1054.780,226.120,-93.750,172.252,35.097,156.574
C07907=1054.786,226.367,-93.778,172.254,35.100,156.575
C07908=1054.793,226.616,-93.805,172.256,35.104,156.576
C07909=1054.799,226.865,-93.831,172.259,35.107,156.576
C07910=1054.805,227.113,-93.859,172.260,35.111,156.577
C07911=1054.811,227.361,-93.886,172.262,35.114,156.578
C07912=1054.818,227.610,-93.914,172.264,35.118,156.579
C07913=1054.825,227.859,-93.940,172.267,35.121,156.579
C07914=1054.831,228.106,-93.967,172.269,35.125,156.580
C07915=1054.837,228.355,-93.994,172.271,35.129,156.581
C07916=1054.843,228.604,-94.021,172.274,35.132,156.581
C07917=1054.850,228.852,-94.049,172.276,35.136,156.582
C07918=1054.856,229.101,-94.076,172.278,35.139,156.583
C07919=1054.862,229.349,-94.103,172.280,35.143,156.584
C07920=1054.869,229.598,-94.130,172.283,35.147,156.584
C07921=1054.875,229.846,-94.157,172.285,35.150,156.585
C07922=1054.881,230.095,-94.184,172.287,35.154,156.586
C07923=1054.887,230.343,-94.212,172.289,35.157,156.586
C07924=1054.894,230.591,-94.240,172.291,35.161,156.587
C07925=1054.900,230.840,-94.267,172.293,35.165,156.588
C07926=1054.906,231.088,-94.294,172.295,35.168,156.589
C07927=1054.912,231.337,-94.322,172.298,35.171,156.589
C07928=1054.919,231.586,-94.349,172.300,35.175,156.590
C07929=1054.925,231.833,-94.377,172.302,35.178,156.591
C07930=1054.931,232.083,-94.404,172.304,35.182,156.591
C07931=1054.937,232.330,-94.431,172.307,35.186,156.592
C07932=1054.944,232.579,-94.459,172.309,35.189,156.593
C07933=1054.950,232.828,-94.486,172.311,35.193,156.594
C07934=1054.956,233.076,-94.513,172.314,35.197,156.594
C07935=1054.962,233.324,-94.541,172.316,35.200,156.595
C07936=1054.969,233.573,-94.569,172.318,35.204,156.596
C07937=1054.975,233.821,-94.596,172.320,35.207,156.596
C07938=1054.981,234.070,-94.624,172.323,35.211,156.597
C07939=1054.987,234.318,-94.652,172.325,35.215,156.598
C07940=1054.993,234.566,-94.679,172.327,35.218,156.599
C07941=1055.000,234.807,-94.706,172.330,35.222,156.599
C07942=1055.005,235.048,-94.732,172.332,35.225,156.600
C07943=1055.012,235.289,-94.759,172.334,35.228,156.601
C07944=1055.018,235.530,-94.786,172.335,35.232,156.601
C07945=1055.024,235.770,-94.812,172.338,35.235,156.602
C07946=1055.029,236.011,-94.840,172.340,35.239,156.603
C07947=1055.036,236.252,-94.866,172.342,35.242,156.603
C07948=1055.042,236.493,-94.893,172.344,35.246,156.604
C07949=1055.048,236.741,-94.921,172.347,35.249,156.605
C07950=1055.054,236.989,-94.949,172.349,35.253,156.606
C07951=1055.061,237.238,-94.976,172.351,35.256,156.606
C07952=1055.067,237.486,-95.005,172.354,35.260,156.607
C07953=1055.074,237.735,-95.032,172.356,35.264,156.608
C07954=1055.080,237.982,-95.060,172.358,35.267,156.608
C07955=1055.086,238.231,-95.088,172.360,35.271,156.609
C07956=1055.092,238.480,-95.116,172.363,35.274,156.610
C07957=1055.099,238.729,-95.143,172.365,35.277,156.611
C07958=1055.106,238.977,-95.170,172.367,35.281,156.611
C07959=1055.111,239.225,-95.198,172.370,35.285,156.612
C07960=1055.118,239.473,-95.227,172.372,35.288,156.613
C07961=1055.125,239.721,-95.255,172.375,35.292,156.613
C07962=1055.130,239.970,-95.283,172.377,35.295,156.614
C07963=1055.137,240.218,-95.310,172.380,35.299,156.615
C07964=1055.143,240.466,-95.338,172.382,35.303,156.616
C07965=1055.149,240.715,-95.366,172.384,35.306,156.616
C07966=1055.156,240.964,-95.394,172.387,35.310,156.617
C07967=1055.162,241.212,-95.422,172.389,35.313,156.618
C07968=1055.168,241.461,-95.450,172.391,35.316,156.618
C07969=1055.175,241.709,-95.477,172.394,35.320,156.619
C07970=1055.181,241.957,-95.506,172.396,35.324,156.620
C07971=1055.187,242.206,-95.534,172.398,35.327,156.621
C07972=1055.193,242.454,-95.563,172.400,35.331,156.621
C07973=1055.200,242.702,-95.590,172.403,35.334,156.622
C07974=1055.205,242.950,-95.618,172.405,35.338,156.623
C07975=1055.211,243.199,-95.647,172.407,35.341,156.623
C07976=1055.218,243.447,-95.675,172.410,35.345,156.624
C07977=1055.224,243.696,-95.703,172.412,35.349,156.625
C07978=1055.231,243.944,-95.731,172.415,35.352,156.626
C07979=1055.237,244.193,-95.759,172.418,35.356,156.626
C07980=1055.243,244.440,-95.787,172.420,35.359,156.627
C07981=1055.249,244.689,-95.816,172.422,35.363,156.628
C07982=1055.255,244.937,-95.844,172.424,35.367,156.629
C07983=1055.262,245.185,-95.873,172.427,35.370,156.629
C07984=1055.268,245.434,-95.901,172.429,35.373,156.630
C07985=1055.275,245.683,-95.929,172.431,35.377,156.631
C07986=1055.281,245.931,-95.958,172.434,35.380,156.631
C07987=1055.287,246.179,-95.986,172.436,35.384,156.632
C07988=1055.293,246.427,-96.013,172.438,35.387,156.633
C07989=1055.299,246.675,-96.042,172.442,35.391,156.634
C07990=1055.305,246.924,-96.071,172.444,35.395,156.634
C07991=1055.312,247.172,-96.100,172.446,35.398,156.635
C07992=1055.318,247.421,-96.128,172.448,35.402,156.636
C07993=1055.324,247.669,-96.157,172.451,35.405,156.636
C07994=1055.330,247.917,-96.185,172.453,35.409,156.637
C07995=1055.336,248.165,-96.214,172.455,35.413,156.638
C07996=1055.342,248.414,-96.242,172.458,35.417,156.639
C07997=1055.348,248.652,-96.269,172.460,35.420,156.639
C07998=1055.354,248.889,-96.297,172.462,35.423,156.640
C07999=1055.360,249.127,-96.325,172.465,35.427,156.641
C08000=1055.366,249.365,-96.352,172.467,35.430,156.642
C08001=1055.371,249.602,-96.379,172.469,35.433,156.642
C08002=1055.377,249.841,-96.406,172.472,35.437,156.643
C08003=1055.384,250.078,-96.434,172.475,35.441,156.644
C08004=1055.390,250.316,-96.461,172.477,35.444,156.644
C08005=1055.396,250.564,-96.490,172.479,35.447,156.645
C08006=1055.402,250.813,-96.519,172.482,35.451,156.646
C08007=1055.408,251.061,-96.548,172.484,35.454,156.646
C08008=1055.415,251.309,-96.576,172.486,35.458,156.647
C08009=1055.421,251.558,-96.605,172.489,35.461,156.648
C08010=1055.427,251.806,-96.634,172.492,35.465,156.649
C08011=1055.434,252.054,-96.663,172.494,35.469,156.649
C08012=1055.439,252.303,-96.691,172.497,35.472,156.650
C08013=1055.446,252.551,-96.720,172.499,35.476,156.651
C08014=1055.452,252.799,-96.749,172.501,35.479,156.652
C08015=1055.458,253.048,-96.777,172.504,35.483,156.652
C08016=1055.465,253.295,-96.806,172.507,35.487,156.653
C08017=1055.471,253.544,-96.835,172.509,35.490,156.654
C08018=1055.477,253.792,-96.864,172.512,35.494,156.654
C08019=1055.484,254.040,-96.893,172.514,35.497,156.655
C08020=1055.490,254.289,-96.921,172.516,35.501,156.656
C08021=1055.496,254.537,-96.950,172.519,35.504,156.657
C08022=1055.502,254.785,-96.979,172.522,35.508,156.657
C08023=1055.508,255.033,-97.008,172.524,35.512,156.658
C08024=1055.515,255.281,-97.037,172.526,35.515,156.659
C08025=1055.521,255.529,-97.066,172.529,35.519,156.660
C08026=1055.527,255.778,-97.095,172.532,35.522,156.660
C08027=1055.534,256.026,-97.124,172.534,35.525,156.661
C08028=1055.541,256.275,-97.153,172.537,35.529,156.662
C08029=1055.547,256.523,-97.182,172.539,35.532,156.662
C08030=1055.553,256.771,-97.211,172.541,35.536,156.663
C08031=1055.559,257.019,-97.240,172.545,35.539,156.664
C08032=1055.566,257.267,-97.269,172.547,35.543,156.665
C08033=1055.572,257.515,-97.298,172.549,35.547,156.665
C08034=1055.578,257.763,-97.327,172.552,35.550,156.666
C08035=1055.585,258.012,-97.356,172.555,35.554,156.667
C08036=1055.591,258.260,-97.385,172.557,35.557,156.668
C08037=1055.597,258.509,-97.414,172.560,35.560,156.668
C08038=1055.604,258.757,-97.443,172.562,35.564,156.669
C08039=1055.610,259.005,-97.472,172.565,35.567,156.670
C08040=1055.617,259.254,-97.502,172.568,35.571,156.670
C08041=1055.623,259.502,-97.531,172.570,35.575,156.671
C08042=1055.630,259.750,-97.559,172.572,35.578,156.672
C08043=1055.636,259.998,-97.588,172.576,35.582,156.673
C08044=1055.643,260.246,-97.617,172.578,35.585,156.673
C08045=1055.649,260.495,-97.647,172.580,35.588,156.674
C08046=1055.656,260.742,-97.677,172.584,35.592,156.675
C08047=1055.662,260.990,-97.706,172.586,35.595,156.675
C08048=1055.668,261.238,-97.735,172.588,35.599,156.676
C08049=1055.675,261.487,-97.764,172.591,35.602,156.677
C08050=1055.682,261.735,-97.793,172.594,35.606,156.678
C08051=1055.688,261.984,-97.822,172.596,35.610,156.678
C08052=1055.694,262.232,-97.851,172.599,35.613,156.679
C08053=1055.701,262.468,-97.880,172.602,35.616,156.680
C08054=1055.707,262.706,-97.908,172.604,35.620,156.680
C08055=1055.713,262.943,-97.936,172.606,35.623,156.681
C08056=1055.719,263.179,-97.964,172.609,35.626,156.682
C08057=1055.725,263.416,-97.992,172.611,35.630,156.682
C08058=1055.731,263.652,-98.020,172.614,35.633,156.683
C08059=1055.737,263.889,-98.048,172.617,35.636,156.684
C08060=1055.743,264.126,-98.076,172.619,35.640,156.685
C08061=1055.750,264.374,-98.106,172.621,35.643,156.685
C08062=1055.755,264.623,-98.136,172.625,35.647,156.686
C08063=1055.762,264.870,-98.166,172.627,35.651,156.687
C08064=1055.768,265.118,-98.195,172.629,35.654,156.688
C08065=1055.774,265.368,-98.225,172.633,35.658,156.688
C08066=1055.781,265.615,-98.254,172.635,35.661,156.689
C08067=1055.787,265.863,-98.283,172.637,35.665,156.690
C08068=1055.793,266.111,-98.314,172.641,35.668,156.690
C08069=1055.800,266.360,-98.343,172.643,35.672,156.691
C08070=1055.806,266.607,-98.373,172.646,35.675,156.692
C08071=1055.812,266.856,-98.403,172.649,35.679,156.693
C08072=1055.819,267.104,-98.433,172.651,35.683,156.693
C08073=1055.825,267.352,-98.462,172.654,35.686,156.694
C08074=1055.831,267.600,-98.492,172.657,35.690,156.695
C08075=1055.838,267.849,-98.521,172.659,35.693,156.696
C08076=1055.844,268.097,-98.552,172.662,35.697,156.696
C08077=1055.850,268.345,-98.581,172.665,35.700,156.697
C08078=1055.857,268.593,-98.611,172.667,35.704,156.698
C08079=1055.863,268.841,-98.641,172.670,35.707,156.699
C08080=1055.869,269.089,-98.670,172.673,35.711,156.699
C08081=1055.876,269.338,-98.701,172.675,35.714,156.700
C08082=1055.882,269.585,-98.731,172.678,35.718,156.701
C08083=1055.888,269.834,-98.761,172.681,35.722,156.702
C08084=1055.895,270.082,-98.791,172.683,35.726,156.702
C08085=1055.901,270.330,-98.821,172.687,35.729,156.703
C08086=1055.907,270.578,-98.850,172.689,35.733,156.704
C08087=1055.913,270.826,-98.881,172.692,35.736,156.705
C08088=1055.920,271.074,-98.910,172.695,35.740,156.705
C08089=1055.926,271.322,-98.941,172.697,35.743,156.706
C08090=1055.932,271.570,-98.970,172.701,35.747,156.707
C08091=1055.939,271.819,-99.001,172.703,35.751,156.708
C08092=1055.945,272.066,-99.031,172.705,35.754,156.708
C08093=1055.952,272.315,-99.061,172.709,35.758,156.709
C08094=1055.958,272.562,-99.091,172.711,35.761,156.710
C08095=1055.964,272.811,-99.121,172.714,35.765,156.711
C08096=1055.970,273.059,-99.151,172.717,35.768,156.711
C08097=1055.977,273.307,-99.181,172.719,35.772,156.712
C08098=1055.983,273.555,-99.212,172.722,35.776,156.713
C08099=1055.989,273.803,-99.242,172.725,35.779,156.714
C08100=1055.996,274.051,-99.272,172.728,35.783,156.714
C08101=1056.002,274.299,-99.303,172.731,35.787,156.715
C08102=1056.008,274.547,-99.333,172.733,35.790,156.716
C08103=1056.015,274.795,-99.363,172.736,35.794,156.717
C08104=1056.021,275.043,-99.394,172.739,35.797,156.717
C08105=1056.027,275.292,-99.424,172.742,35.801,156.718
C08106=1056.034,275.539,-99.454,172.744,35.804,156.719
C08107=1056.040,275.788,-99.485,172.748,35.808,156.720
C08108=1056.046,276.035,-99.515,172.750,35.812,156.720
C08109=1056.053,276.275,-99.544,172.753,35.815,156.721
C08110=1056.059,276.513,-99.573,172.756,35.818,156.722
C08111=1056.064,276.752,-99.603,172.758,35.822,156.723
C08112=1056.071,276.991,-99.632,172.761,35.825,156.723
C08113=1056.077,277.229,-99.661,172.764,35.829,156.724
C08114=1056.083,277.468,-99.691,172.766,35.832,156.725
C08115=1056.089,277.707,-99.720,172.770,35.836,156.726
C08116=1056.095,277.946,-99.749,172.772,35.840,156.726
C08117=1056.102,278.194,-99.780,172.774,35.843,156.727
C08118=1056.108,278.442,-99.810,172.778,35.847,156.728
C08119=1056.114,278.690,-99.842,172.780,35.850,156.729
C08120=1056.121,278.939,-99.872,172.784,35.854,156.729
C08121=1056.127,279.186,-99.902,172.786,35.858,156.730
C08122=1056.134,279.435,-99.933,172.789,35.861,156.731
C08123=1056.140,279.682,-99.963,172.792,35.865,156.732
C08124=1056.146,279.930,-99.995,172.795,35.868,156.732
C08125=1056.152,280.178,-100.025,172.797,35.872,156.733
C08126=1056.159,280.427,-100.056,172.801,35.876,156.734
C08127=1056.165,280.675,-100.087,172.803,35.880,156.735
C08128=1056.171,280.922,-100.118,172.807,35.883,156.735
C08129=1056.177,281.171,-100.148,172.809,35.887,156.736
C08130=1056.184,281.418,-100.179,172.812,35.891,156.737
C08131=1056.190,281.667,-100.210,172.815,35.894,156.738
C08132=1056.197,281.915,-100.242,172.818,35.898,156.739
C08133=1056.203,282.162,-100.272,172.821,35.901,156.739
C08134=1056.209,282.411,-100.303,172.824,35.905,156.740
C08135=1056.215,282.658,-100.334,172.826,35.909,156.741
C08136=1056.222,282.907,-100.364,172.830,35.912,156.742
C08137=1056.228,283.154,-100.396,172.832,35.916,156.742
C08138=1056.234,283.402,-100.426,172.836,35.920,156.743
C08139=1056.241,283.650,-100.458,172.838,35.924,156.744
C08140=1056.247,283.899,-100.488,172.841,35.927,156.745
C08141=1056.253,284.146,-100.519,172.845,35.931,156.746
C08142=1056.260,284.394,-100.550,172.847,35.935,156.746
C08143=1056.266,284.642,-100.582,172.851,35.938,156.747
C08144=1056.272,284.890,-100.612,172.853,35.942,156.748
C08145=1056.279,285.138,-100.643,172.856,35.945,156.749
C08146=1056.286,285.386,-100.675,172.859,35.949,156.750
C08147=1056.292,285.634,-100.705,172.862,35.953,156.750
C08148=1056.298,285.882,-100.737,172.864,35.956,156.751
C08149=1056.305,286.130,-100.768,172.868,35.960,156.752
C08150=1056.311,286.378,-100.799,172.871,35.964,156.753
C08151=1056.318,286.625,-100.830,172.874,35.968,156.753
C08152=1056.324,286.873,-100.861,172.877,35.971,156.754
C08153=1056.331,287.122,-100.892,172.879,35.975,156.755
C08154=1056.337,287.370,-100.923,172.883,35.979,156.756
C08155=1056.344,287.617,-100.954,172.886,35.982,156.757
C08156=1056.350,287.865,-100.985,172.889,35.986,156.757
C08157=1056.356,288.114,-101.017,172.892,35.989,156.758
C08158=1056.363,288.361,-101.049,172.895,35.993,156.759
C08159=1056.369,288.609,-101.080,172.898,35.997,156.760
C08160=1056.376,288.857,-101.111,172.900,36.000,156.760
C08161=1056.381,289.105,-101.142,172.904,36.004,156.761
C08162=1056.388,289.353,-101.174,172.907,36.008,156.762
C08163=1056.395,289.601,-101.205,172.910,36.011,156.763
C08164=1056.401,289.848,-101.236,172.913,36.016,156.764
C08165=1056.407,290.093,-101.267,172.915,36.019,156.764
C08166=1056.413,290.337,-101.299,172.919,36.023,156.765
C08167=1056.420,290.581,-101.330,172.922,36.027,156.766
C08168=1056.426,290.826,-101.360,172.925,36.030,156.767
C08169=1056.432,291.070,-101.391,172.928,36.034,156.768
C08170=1056.438,291.314,-101.423,172.931,36.038,156.768
C08171=1056.445,291.559,-101.454,172.934,36.041,156.769
C08172=1056.451,291.803,-101.485,172.937,36.045,156.770
C08173=1056.457,292.051,-101.516,172.940,36.049,156.771
C08174=1056.463,292.299,-101.548,172.943,36.052,156.772
C08175=1056.470,292.547,-101.580,172.947,36.056,156.772
C08176=1056.477,292.795,-101.611,172.949,36.060,156.773
C08177=1056.483,293.043,-101.643,172.952,36.063,156.774
C08178=1056.490,293.291,-101.675,172.956,36.068,156.775
C08179=1056.497,293.538,-101.707,172.958,36.071,156.776
C08180=1056.503,293.786,-101.739,172.962,36.075,156.776
C08181=1056.509,294.033,-101.770,172.965,36.079,156.777
C08182=1056.515,294.281,-101.801,172.968,36.082,156.778
C08183=1056.521,294.529,-101.833,172.971,36.086,156.779
C08184=1056.528,294.777,-101.865,172.974,36.090,156.780
C08185=1056.534,295.025,-101.898,172.977,36.094,156.780
C08186=1056.541,295.273,-101.929,172.980,36.097,156.781
C08187=1056.547,295.521,-101.961,172.984,36.101,156.782
C08188=1056.554,295.769,-101.992,172.986,36.105,156.783
C08189=1056.560,296.017,-102.025,172.990,36.109,156.784
C08190=1056.567,296.265,-102.057,172.993,36.112,156.784
C08191=1056.573,296.513,-102.089,172.996,36.116,156.785
C08192=1056.580,296.761,-102.120,172.999,36.120,156.786
C08193=1056.586,297.008,-102.153,173.002,36.124,156.787
C08194=1056.592,297.256,-102.185,173.005,36.128,156.788
C08195=1056.598,297.503,-102.217,173.008,36.132,156.789
C08196=1056.604,297.751,-102.249,173.012,36.136,156.790
C08197=1056.611,297.999,-102.281,173.015,36.140,156.790
C08198=1056.617,298.247,-102.313,173.018,36.143,156.791
C08199=1056.624,298.494,-102.346,173.021,36.147,156.792
C08200=1056.630,298.743,-102.378,173.025,36.151,156.793
C08201=1056.636,298.990,-102.410,173.027,36.155,156.794
C08202=1056.642,299.238,-102.442,173.030,36.159,156.795
C08203=1056.648,299.486,-102.475,173.034,36.163,156.795
C08204=1056.655,299.734,-102.507,173.036,36.166,156.796
C08205=1056.661,299.981,-102.539,173.040,36.171,156.797
C08206=1056.667,300.230,-102.571,173.043,36.175,156.798
C08207=1056.674,300.477,-102.604,173.047,36.178,156.799
C08208=1056.680,300.725,-102.637,173.049,36.182,156.800
C08209=1056.687,300.973,-102.668,173.053,36.186,156.801
C08210=1056.693,301.220,-102.701,173.056,36.190,156.801
C08211=1056.699,301.468,-102.734,173.060,36.194,156.802
C08212=1056.705,301.716,-102.766,173.062,36.198,156.803
C08213=1056.711,301.964,-102.799,173.066,36.202,156.804
C08214=1056.718,302.211,-102.831,173.069,36.205,156.805
C08215=1056.724,302.459,-102.863,173.072,36.209,156.806
C08216=1056.731,302.707,-102.895,173.076,36.213,156.806
C08217=1056.737,302.954,-102.928,173.078,36.217,156.807
C08218=1056.744,303.203,-102.961,173.082,36.221,156.808
C08219=1056.750,303.451,-102.993,173.085,36.225,156.809
C08220=1056.757,303.698,-103.025,173.089,36.229,156.810
C08221=1056.764,303.955,-103.059,173.092,36.233,156.811
C08222=1056.769,304.210,-103.093,173.095,36.237,156.812
C08223=1056.776,304.467,-103.127,173.098,36.241,156.813
C08224=1056.783,304.724,-103.161,173.102,36.245,156.813
C08225=1056.789,304.971,-103.193,173.105,36.249,156.814
C08226=1056.796,305.219,-103.225,173.109,36.253,156.815
C08227=1056.803,305.467,-103.259,173.112,36.257,156.816
C08228=1056.809,305.715,-103.291,173.116,36.261,156.817
C08229=1056.816,305.962,-103.324,173.118,36.264,156.818
C08230=1056.822,306.210,-103.357,173.122,36.268,156.818
C08231=1056.828,306.457,-103.389,173.125,36.273,156.819
C08232=1056.835,306.706,-103.423,173.129,36.277,156.820
C08233=1056.842,306.953,-103.455,173.132,36.280,156.821
C08234=1056.848,307.200,-103.487,173.136,36.284,156.822
C08235=1056.855,307.448,-103.520,173.138,36.288,156.823
C08236=1056.862,307.696,-103.553,173.142,36.292,156.824
C08237=1056.868,307.944,-103.586,173.145,36.296,156.825
C08238=1056.874,308.192,-103.619,173.149,36.300,156.825
C08239=1056.880,308.439,-103.652,173.152,36.304,156.826
C08240=1056.887,308.687,-103.685,173.156,36.308,156.827
C08241=1056.894,308.935,-103.717,173.159,36.312,156.828
C08242=1056.901,309.182,-103.750,173.163,36.316,156.829
C08243=1056.908,309.430,-103.783,173.165,36.320,156.830
C08244=1056.914,309.678,-103.816,173.168,36.323,156.831
C08245=1056.920,309.925,-103.849,173.172,36.327,156.831
C08246=1056.927,310.173,-103.882,173.176,36.331,156.832
C08247=1056.934,310.421,-103.915,173.179,36.335,156.833
C08248=1056.940,310.668,-103.948,173.183,36.340,156.834
C08249=1056.947,310.916,-103.981,173.186,36.344,156.835
C08250=1056.953,311.164,-104.014,173.189,36.347,156.836
C08251=1056.960,311.412,-104.047,173.193,36.351,156.837
C08252=1056.967,311.659,-104.081,173.196,36.355,156.838
C08253=1056.973,311.907,-104.113,173.199,36.359,156.838
C08254=1056.980,312.155,-104.146,173.203,36.363,156.839
C08255=1056.987,312.402,-104.180,173.206,36.367,156.840
C08256=1056.994,312.650,-104.213,173.210,36.371,156.841
C08257=1057.000,312.898,-104.246,173.213,36.375,156.842
C08258=1057.008,313.145,-104.279,173.216,36.379,156.843
C08259=1057.014,313.393,-104.312,173.220,36.383,156.844
C08260=1057.020,313.642,-104.345,173.224,36.387,156.845
C08261=1057.027,313.888,-104.379,173.227,36.391,156.846
C08262=1057.033,314.136,-104.413,173.231,36.395,156.847
C08263=1057.040,314.384,-104.446,173.234,36.399,156.847
C08264=1057.046,314.631,-104.480,173.238,36.403,156.848
C08265=1057.052,314.879,-104.513,173.241,36.407,156.849
C08266=1057.058,315.127,-104.547,173.245,36.412,156.850
C08267=1057.065,315.374,-104.581,173.247,36.416,156.851
C08268=1057.071,315.621,-104.613,173.251,36.420,156.852
C08269=1057.078,315.869,-104.648,173.254,36.424,156.853
C08270=1057.084,316.117,-104.681,173.258,36.428,156.854
C08271=1057.090,316.365,-104.715,173.261,36.433,156.855
C08272=1057.097,316.612,-104.749,173.265,36.437,156.856
C08273=1057.103,316.860,-104.783,173.269,36.441,156.857
C08274=1057.110,317.108,-104.816,173.272,36.445,156.858
C08275=1057.116,317.356,-104.850,173.276,36.449,156.859
C08276=1057.123,317.603,-104.884,173.279,36.453,156.859
C08277=1057.129,317.864,-104.920,173.283,36.458,156.860
C08278=1057.136,318.124,-104.955,173.286,36.462,156.861
C08279=1057.143,318.385,-104.991,173.290,36.467,156.862
C08280=1057.149,318.645,-105.026,173.295,36.471,156.863
C08281=1057.157,318.892,-105.060,173.298,36.475,156.864
C08282=1057.163,319.140,-105.094,173.302,36.479,156.865
C08283=1057.169,319.388,-105.128,173.305,36.483,156.866
C08284=1057.176,319.635,-105.162,173.309,36.488,156.867
C08285=1057.182,319.883,-105.195,173.312,36.492,156.868
C08286=1057.189,320.131,-105.229,173.316,36.496,156.869
C08287=1057.195,320.378,-105.263,173.319,36.500,156.870
C08288=1057.202,320.626,-105.297,173.323,36.504,156.871
C08289=1057.208,320.873,-105.331,173.326,36.508,156.872
C08290=1057.215,321.121,-105.365,173.330,36.513,156.873
C08291=1057.222,321.369,-105.399,173.334,36.517,156.874
C08292=1057.228,321.616,-105.433,173.337,36.521,156.875
C08293=1057.235,321.864,-105.467,173.341,36.526,156.876
C08294=1057.241,322.112,-105.502,173.344,36.530,156.877
C08295=1057.248,322.359,-105.535,173.348,36.534,156.878
C08296=1057.254,322.606,-105.570,173.351,36.538,156.878
C08297=1057.262,322.854,-105.604,173.355,36.542,156.879
C08298=1057.268,323.101,-105.638,173.359,36.547,156.880
C08299=1057.274,323.349,-105.672,173.362,36.551,156.881
C08300=1057.281,323.597,-105.706,173.366,36.555,156.882
C08301=1057.288,323.845,-105.741,173.369,36.559,156.883
C08302=1057.294,324.092,-105.774,173.373,36.563,156.884
C08303=1057.301,324.339,-105.809,173.376,36.568,156.885
C08304=1057.308,324.587,-105.843,173.380,36.572,156.886
C08305=1057.315,324.835,-105.878,173.385,36.576,156.887
C08306=1057.321,325.082,-105.912,173.388,36.580,156.888
C08307=1057.328,325.329,-105.946,173.392,36.585,156.889
C08308=1057.334,325.577,-105.981,173.395,36.589,156.890
C08309=1057.341,325.825,-106.015,173.399,36.594,156.891
C08310=1057.348,326.073,-106.049,173.403,36.598,156.892
C08311=1057.354,326.319,-106.084,173.406,36.602,156.893
C08312=1057.362,326.567,-106.117,173.410,36.606,156.894
C08313=1057.368,326.815,-106.152,173.413,36.611,156.895
C08314=1057.375,327.062,-106.187,173.418,36.615,156.896
C08315=1057.382,327.310,-106.221,173.422,36.619,156.897
C08316=1057.389,327.558,-106.256,173.425,36.623,156.898
C08317=1057.395,327.805,-106.290,173.429,36.628,156.899
C08318=1057.403,328.053,-106.325,173.432,36.632,156.900
C08319=1057.409,328.300,-106.359,173.436,36.636,156.901
C08320=1057.415,328.547,-106.394,173.441,36.641,156.902
C08321=1057.423,328.795,-106.428,173.444,36.645,156.903
C08322=1057.429,329.042,-106.463,173.448,36.649,156.904
C08323=1057.436,329.290,-106.497,173.451,36.653,156.905
C08324=1057.443,329.537,-106.532,173.455,36.658,156.906
C08325=1057.450,329.785,-106.566,173.459,36.662,156.907
C08326=1057.456,330.033,-106.602,173.463,36.666,156.908
C08327=1057.464,330.280,-106.635,173.467,36.671,156.909
C08328=1057.470,330.528,-106.671,173.470,36.676,156.910
C08329=1057.477,330.775,-106.706,173.474,36.680,156.911
C08330=1057.483,331.023,-106.741,173.478,36.684,156.912
C08331=1057.490,331.271,-106.776,173.481,36.689,156.913
C08332=1057.496,331.518,-106.811,173.486,36.693,156.914
C08333=1057.503,331.773,-106.847,173.490,36.698,156.915
C08334=1057.511,332.028,-106.883,173.493,36.702,156.916
C08335=1057.518,332.283,-106.919,173.498,36.707,156.917
C08336=1057.524,332.538,-106.954,173.502,36.712,156.918
C08337=1057.531,332.785,-106.989,173.505,36.716,156.919
C08338=1057.538,333.033,-107.025,173.509,36.721,156.920
C08339=1057.544,333.280,-107.060,173.513,36.725,156.921
C08340=1057.550,333.528,-107.095,173.517,36.729,156.922
C08341=1057.557,333.775,-107.131,173.521,36.734,156.923
C08342=1057.564,334.023,-107.166,173.524,36.738,156.924
C08343=1057.571,334.271,-107.201,173.528,36.743,156.925
C08344=1057.578,334.518,-107.236,173.533,36.748,156.926
C08345=1057.585,334.765,-107.271,173.536,36.752,156.927
C08346=1057.592,335.013,-107.307,173.540,36.757,156.928
C08347=1057.598,335.260,-107.342,173.544,36.761,156.929
C08348=1057.605,335.507,-107.377,173.548,36.766,156.930
C08349=1057.612,335.755,-107.412,173.552,36.770,156.931
C08350=1057.619,336.002,-107.447,173.556,36.775,156.932
C08351=1057.625,336.250,-107.483,173.559,36.780,156.934
C08352=1057.631,336.497,-107.518,173.564,36.784,156.935
C08353=1057.639,336.745,-107.554,173.568,36.789,156.936
C08354=1057.646,336.992,-107.589,173.571,36.793,156.937
C08355=1057.653,337.239,-107.624,173.576,36.798,156.938
C08356=1057.659,337.487,-107.660,173.580,36.802,156.939
C08357=1057.665,337.734,-107.695,173.583,36.807,156.940
C08358=1057.672,337.981,-107.731,173.587,36.812,156.941
C08359=1057.679,338.229,-107.767,173.592,36.817,156.942
C08360=1057.685,338.476,-107.802,173.596,36.821,156.943
C08361=1057.693,338.724,-107.838,173.599,36.826,156.944
C08362=1057.699,338.971,-107.874,173.604,36.831,156.945
C08363=1057.706,339.219,-107.909,173.608,36.835,156.946
C08364=1057.713,339.465,-107.945,173.611,36.840,156.947
C08365=1057.719,339.713,-107.981,173.616,36.845,156.949
C08366=1057.726,339.961,-108.016,173.620,36.849,156.950
C08367=1057.733,340.208,-108.052,173.623,36.854,156.951
C08368=1057.739,340.456,-108.088,173.628,36.859,156.952
C08369=1057.746,340.702,-108.124,173.632,36.863,156.953
C08370=1057.754,340.950,-108.159,173.636,36.868,156.954
C08371=1057.760,341.197,-108.196,173.640,36.873,156.955
C08372=1057.767,341.445,-108.231,173.644,36.877,156.956
C08373=1057.773,341.692,-108.267,173.648,36.882,156.957
C08374=1057.781,341.939,-108.303,173.652,36.887,156.958
C08375=1057.788,342.187,-108.339,173.656,36.892,156.959
C08376=1057.794,342.434,-108.375,173.661,36.897,156.961
C08377=1057.801,342.682,-108.410,173.665,36.901,156.962
C08378=1057.808,342.929,-108.446,173.668,36.906,156.963
C08379=1057.815,343.176,-108.483,173.673,36.911,156.964
C08380=1057.822,343.424,-108.518,173.677,36.916,156.965
C08381=1057.828,343.671,-108.555,173.680,36.920,156.966
C08382=1057.835,343.918,-108.591,173.685,36.925,156.967
C08383=1057.842,344.165,-108.627,173.689,36.930,156.969
C08384=1057.849,344.413,-108.663,173.694,36.935,156.970
C08385=1057.856,344.660,-108.699,173.697,36.940,156.971
C08386=1057.863,344.907,-108.736,173.701,36.944,156.972
C08387=1057.869,345.154,-108.772,173.706,36.949,156.973
C08388=1057.877,345.402,-108.808,173.710,36.954,156.974
C08389=1057.883,345.653,-108.845,173.715,36.960,156.975
C08390=1057.890,345.903,-108.882,173.718,36.964,156.976
C08391=1057.897,346.154,-108.919,173.723,36.969,156.978
C08392=1057.904,346.405,-108.955,173.727,36.974,156.979
C08393=1057.911,346.653,-108.992,173.732,36.979,156.980
C08394=1057.918,346.899,-109.028,173.735,36.984,156.981
C08395=1057.925,347.147,-109.065,173.740,36.989,156.982
C08396=1057.931,347.394,-109.101,173.744,36.994,156.983
C08397=1057.938,347.642,-109.138,173.748,36.999,156.985
C08398=1057.945,347.888,-109.175,173.752,37.004,156.986
C08399=1057.952,348.135,-109.211,173.756,37.009,156.987
C08400=1057.959,348.383,-109.248,173.761,37.014,156.988
C08401=1057.966,348.630,-109.284,173.765,37.019,156.989
C08402=1057.973,348.877,-109.320,173.770,37.024,156.991
C08403=1057.979,349.125,-109.357,173.773,37.028,156.992
C08404=1057.986,349.372,-109.394,173.778,37.033,156.993
C08405=1057.994,349.619,-109.431,173.782,37.039,156.994
C08406=1058.000,349.866,-109.467,173.787,37.044,156.995
C08407=1058.007,350.114,-109.504,173.790,37.049,156.996
C08408=1058.014,350.360,-109.541,173.795,37.054,156.998
C08409=1058.021,350.608,-109.577,173.799,37.059,156.999
C08410=1058.028,350.856,-109.614,173.804,37.064,157.000
C08411=1058.035,351.103,-109.651,173.809,37.069,157.001
C08412=1058.042,351.350,-109.688,173.813,37.074,157.002
C08413=1058.048,351.597,-109.725,173.817,37.079,157.004
C08414=1058.055,351.844,-109.762,173.821,37.084,157.005
C08415=1058.063,352.091,-109.798,173.826,37.089,157.006
C08416=1058.070,352.338,-109.835,173.830,37.094,157.007
C08417=1058.077,352.586,-109.872,173.835,37.099,157.008
C08418=1058.083,352.832,-109.909,173.839,37.105,157.010
C08419=1058.090,353.080,-109.946,173.843,37.110,157.011
C08420=1058.098,353.327,-109.984,173.847,37.115,157.012
C08421=1058.104,353.574,-110.020,173.852,37.120,157.013
C08422=1058.111,353.821,-110.058,173.857,37.126,157.015
C08423=1058.118,354.068,-110.095,173.861,37.131,157.016
C08424=1058.125,354.315,-110.132,173.866,37.136,157.017
C08425=1058.132,354.562,-110.169,173.869,37.141,157.018
C08426=1058.139,354.809,-110.207,173.874,37.146,157.020
C08427=1058.146,355.057,-110.244,173.879,37.151,157.021
C08428=1058.153,355.304,-110.281,173.883,37.157,157.022
C08429=1058.160,355.551,-110.318,173.888,37.162,157.023
C08430=1058.167,355.798,-110.356,173.892,37.167,157.025
C08431=1058.175,356.045,-110.393,173.897,37.172,157.026
C08432=1058.181,356.292,-110.430,173.901,37.177,157.027
C08433=1058.188,356.539,-110.467,173.905,37.183,157.028
C08434=1058.195,356.786,-110.505,173.910,37.188,157.030
C08435=1058.203,357.034,-110.542,173.915,37.193,157.031
C08436=1058.209,357.281,-110.580,173.919,37.198,157.032
C08437=1058.216,357.527,-110.618,173.924,37.204,157.033
C08438=1058.223,357.775,-110.655,173.929,37.210,157.035
C08439=1058.230,358.022,-110.693,173.933,37.215,157.036
C08440=1058.237,358.269,-110.730,173.937,37.220,157.037
C08441=1058.245,358.516,-110.768,173.942,37.225,157.039
C08442=1058.252,358.763,-110.805,173.946,37.231,157.040
C08443=1058.258,359.010,-110.843,173.951,37.236,157.041
C08444=1058.265,359.257,-110.881,173.956,37.242,157.043
C08445=1058.277,359.666,-110.943,173.964,37.251,157.045
C08446=1058.288,360.074,-111.005,173.971,37.259,157.047
C08447=1058.301,360.482,-111.068,173.979,37.268,157.049
C08448=1058.312,360.891,-111.131,173.986,37.277,157.051
C08449=1058.319,361.138,-111.168,173.991,37.283,157.052
C08450=1058.326,361.384,-111.206,173.995,37.288,157.054
C08451=1058.334,361.631,-111.244,174.000,37.294,157.055
C08452=1058.340,361.879,-111.282,174.005,37.299,157.056
C08453=1058.348,362.125,-111.320,174.010,37.305,157.058
C08454=1058.355,362.372,-111.357,174.014,37.310,157.059
C08455=1058.362,362.619,-111.396,174.019,37.316,157.060
C08456=1058.369,362.866,-111.434,174.024,37.321,157.062
C08457=1058.376,363.113,-111.472,174.029,37.327,157.063
C08458=1058.384,363.361,-111.511,174.034,37.333,157.064
C08459=1058.391,363.608,-111.548,174.038,37.338,157.066
C08460=1058.398,363.855,-111.586,174.042,37.344,157.067
C08461=1058.405,364.101,-111.625,174.048,37.350,157.069
C08462=1058.412,364.349,-111.663,174.053,37.355,157.070
C08463=1058.419,364.595,-111.702,174.056,37.361,157.071
C08464=1058.427,364.842,-111.740,174.061,37.366,157.073
C08465=1058.433,365.089,-111.778,174.066,37.372,157.074
C08466=1058.440,365.336,-111.817,174.071,37.378,157.075
C08467=1058.448,365.583,-111.855,174.076,37.383,157.077
C08468=1058.454,365.830,-111.893,174.080,37.389,157.078
C08469=1058.462,366.077,-111.931,174.085,37.395,157.080
C08470=1058.469,366.323,-111.970,174.091,37.401,157.081
C08471=1058.476,366.570,-112.008,174.095,37.406,157.082
C08472=1058.484,366.817,-112.048,174.100,37.412,157.084
C08473=1058.490,367.064,-112.086,174.106,37.418,157.085
C08474=1058.498,367.311,-112.124,174.109,37.424,157.087
C08475=1058.504,367.558,-112.163,174.115,37.430,157.088
C08476=1058.512,367.805,-112.201,174.120,37.435,157.090
C08477=1058.522,368.145,-112.255,174.126,37.443,157.092
C08478=1058.532,368.487,-112.309,174.133,37.452,157.094
C08479=1058.541,368.828,-112.362,174.140,37.459,157.095
C08480=1058.551,369.168,-112.416,174.147,37.467,157.097
C08481=1058.560,369.416,-112.454,174.151,37.474,157.099
C08482=1058.566,369.663,-112.493,174.156,37.479,157.100
C08483=1058.573,369.909,-112.532,174.161,37.485,157.102
C08484=1058.581,370.157,-112.571,174.167,37.491,157.103
C08485=1058.588,370.403,-112.609,174.172,37.497,157.105
C08486=1058.595,370.650,-112.648,174.177,37.503,157.106
C08487=1058.603,370.896,-112.687,174.182,37.509,157.108
C08488=1058.610,371.144,-112.726,174.187,37.515,157.109
C08489=1058.618,371.390,-112.765,174.192,37.521,157.111
C08490=1058.626,371.637,-112.805,174.197,37.526,157.112
C08491=1058.632,371.884,-112.843,174.202,37.532,157.113
C08492=1058.640,372.130,-112.882,174.207,37.538,157.115
C08493=1058.648,372.377,-112.922,174.212,37.544,157.116
C08494=1058.654,372.624,-112.960,174.217,37.550,157.118
C08495=1058.662,372.870,-113.000,174.222,37.556,157.119
C08496=1058.669,373.118,-113.039,174.228,37.562,157.121
C08497=1058.677,373.392,-113.083,174.233,37.569,157.123
C08498=1058.685,373.665,-113.127,174.238,37.576,157.124
C08499=1058.692,373.940,-113.170,174.244,37.583,157.126
C08500=1058.701,374.214,-113.214,174.250,37.590,157.128
C08501=1058.709,374.460,-113.253,174.255,37.596,157.129
C08502=1058.716,374.707,-113.293,174.260,37.602,157.131
C08503=1058.723,374.953,-113.332,174.265,37.608,157.132
C08504=1058.730,375.200,-113.372,174.270,37.614,157.134
C08505=1058.738,375.447,-113.411,174.275,37.621,157.135
C08506=1058.745,375.694,-113.450,174.280,37.627,157.137
C08507=1058.752,375.940,-113.490,174.286,37.633,157.138
C08508=1058.760,376.187,-113.530,174.292,37.639,157.140
C08509=1058.767,376.433,-113.570,174.297,37.645,157.142
C08510=1058.775,376.680,-113.609,174.302,37.652,157.143
C08511=1058.782,376.927,-113.649,174.307,37.658,157.145
C08512=1058.789,377.174,-113.688,174.313,37.664,157.146
C08513=1058.797,377.421,-113.728,174.318,37.670,157.148
C08514=1058.804,377.667,-113.768,174.323,37.677,157.149
C08515=1058.812,377.914,-113.808,174.328,37.683,157.151
C08516=1058.819,378.161,-113.848,174.333,37.690,157.153
C08517=1058.827,378.407,-113.887,174.339,37.696,157.154
C08518=1058.834,378.654,-113.927,174.344,37.702,157.156
C08519=1058.841,378.900,-113.967,174.350,37.709,157.157
C08520=1058.849,379.147,-114.006,174.355,37.715,157.159
C08521=1058.857,379.393,-114.047,174.360,37.722,157.161
C08522=1058.865,379.640,-114.087,174.366,37.728,157.162
C08523=1058.872,379.887,-114.127,174.371,37.734,157.164
C08524=1058.880,380.134,-114.166,174.376,37.741,157.165
C08525=1058.887,380.380,-114.206,174.381,37.747,157.167
C08526=1058.895,380.627,-114.248,174.388,37.754,157.169
C08527=1058.902,380.873,-114.287,174.393,37.760,157.170
C08528=1058.910,381.120,-114.327,174.398,37.767,157.172
C08529=1058.917,381.367,-114.368,174.403,37.773,157.174
C08530=1058.924,381.613,-114.408,174.409,37.780,157.175
C08531=1058.932,381.860,-114.448,174.414,37.786,157.177
C08532=1058.939,382.106,-114.489,174.420,37.793,157.179
C08533=1058.947,382.353,-114.529,174.426,37.800,157.180
C08534=1058.954,382.599,-114.569,174.431,37.806,157.182
C08535=1058.961,382.846,-114.610,174.436,37.813,157.184
C08536=1058.969,383.092,-114.650,174.441,37.819,157.185
C08537=1058.977,383.339,-114.691,174.448,37.826,157.187
C08538=1058.984,383.586,-114.732,174.453,37.833,157.189
C08539=1058.992,383.831,-114.772,174.458,37.839,157.190
C08540=1058.998,384.079,-114.812,174.464,37.846,157.192
C08541=1059.007,384.325,-114.853,174.470,37.853,157.194
C08542=1059.015,384.571,-114.894,174.475,37.860,157.196
C08543=1059.022,384.818,-114.935,174.481,37.866,157.197
C08544=1059.030,385.065,-114.975,174.486,37.874,157.199
C08545=1059.037,385.311,-115.016,174.492,37.880,157.201
C08546=1059.045,385.558,-115.057,174.498,37.887,157.203
C08547=1059.053,385.804,-115.097,174.503,37.894,157.204
C08548=1059.060,386.051,-115.138,174.509,37.901,157.206
C08549=1059.068,386.296,-115.179,174.515,37.908,157.208
C08550=1059.075,386.543,-115.220,174.520,37.914,157.209
C08551=1059.083,386.789,-115.261,174.527,37.921,157.211
C08552=1059.091,387.036,-115.302,174.532,37.928,157.213
C08553=1059.100,387.341,-115.352,174.539,37.937,157.215
C08554=1059.110,387.647,-115.403,174.546,37.945,157.217
C08555=1059.119,387.951,-115.454,174.553,37.954,157.220
C08556=1059.129,388.257,-115.504,174.561,37.963,157.222
C08557=1059.137,388.503,-115.546,174.566,37.970,157.224
C08558=1059.145,388.749,-115.586,174.572,37.977,157.226
C08559=1059.152,388.996,-115.628,174.578,37.984,157.227
C08560=1059.161,389.243,-115.669,174.584,37.991,157.229
C08561=1059.168,389.490,-115.710,174.590,37.998,157.231
C08562=1059.176,389.735,-115.751,174.596,38.005,157.233
C08563=1059.184,389.982,-115.792,174.601,38.012,157.235
C08564=1059.192,390.228,-115.833,174.607,38.019,157.236
C08565=1059.199,390.474,-115.875,174.613,38.026,157.238
C08566=1059.207,390.721,-115.917,174.619,38.033,157.240
C08567=1059.215,390.967,-115.959,174.625,38.040,157.242
C08568=1059.223,391.214,-115.999,174.631,38.047,157.244
C08569=1059.230,391.460,-116.041,174.637,38.055,157.246
C08570=1059.238,391.706,-116.082,174.643,38.061,157.247
C08571=1059.247,391.953,-116.124,174.649,38.069,157.249
C08572=1059.254,392.199,-116.165,174.655,38.076,157.251
C08573=1059.262,392.445,-116.207,174.661,38.084,157.253
C08574=1059.269,392.691,-116.249,174.668,38.091,157.255
C08575=1059.278,392.938,-116.290,174.673,38.098,157.257
C08576=1059.285,393.184,-116.332,174.680,38.105,157.259
C08577=1059.293,393.430,-116.374,174.685,38.113,157.261
C08578=1059.301,393.677,-116.416,174.692,38.120,157.263
C08579=1059.308,393.923,-116.458,174.697,38.127,157.265
C08580=1059.316,394.169,-116.500,174.704,38.135,157.267
C08581=1059.324,394.416,-116.542,174.709,38.142,157.268
C08582=1059.333,394.662,-116.583,174.716,38.150,157.270
C08583=1059.340,394.908,-116.625,174.722,38.157,157.272
C08584=1059.348,395.154,-116.667,174.728,38.165,157.274
C08585=1059.356,395.400,-116.709,174.735,38.172,157.276
C08586=1059.364,395.647,-116.752,174.740,38.180,157.278
C08587=1059.372,395.893,-116.794,174.747,38.187,157.280
C08588=1059.380,396.140,-116.836,174.753,38.195,157.282
C08589=1059.388,396.386,-116.878,174.759,38.202,157.284
C08590=1059.396,396.632,-116.920,174.766,38.210,157.286
C08591=1059.403,396.878,-116.962,174.772,38.218,157.288
C08592=1059.412,397.124,-117.005,174.778,38.225,157.290
C08593=1059.419,397.370,-117.047,174.784,38.233,157.292
C08594=1059.428,397.617,-117.089,174.791,38.241,157.294
C08595=1059.435,397.863,-117.131,174.797,38.248,157.296
C08596=1059.444,398.109,-117.174,174.803,38.256,157.298
C08597=1059.451,398.355,-117.216,174.810,38.264,157.300
C08598=1059.460,398.602,-117.259,174.816,38.272,157.302
C08599=1059.468,398.848,-117.302,174.822,38.280,157.304
C08600=1059.475,399.094,-117.344,174.829,38.287,157.306
C08601=1059.483,399.340,-117.387,174.835,38.295,157.309
C08602=1059.492,399.587,-117.430,174.841,38.303,157.311
C08603=1059.499,399.832,-117.472,174.848,38.311,157.313
C08604=1059.508,400.079,-117.515,174.855,38.318,157.315
C08605=1059.516,400.325,-117.558,174.861,38.326,157.317
C08606=1059.523,400.570,-117.601,174.867,38.334,157.319
C08607=1059.532,400.817,-117.643,174.874,38.342,157.321
C08608=1059.540,401.063,-117.686,174.881,38.350,157.323
C08609=1059.551,401.386,-117.742,174.889,38.361,157.326
C08610=1059.561,401.708,-117.799,174.897,38.372,157.329
C08611=1059.572,402.031,-117.855,174.907,38.382,157.331
C08612=1059.583,402.353,-117.911,174.915,38.392,157.334
C08613=1059.591,402.600,-117.954,174.922,38.401,157.337
C08614=1059.599,402.846,-117.997,174.929,38.409,157.339
C08615=1059.608,403.092,-118.040,174.936,38.417,157.341
C08616=1059.615,403.338,-118.084,174.941,38.425,157.343
C08617=1059.624,403.584,-118.127,174.948,38.433,157.345
C08618=1059.632,403.830,-118.170,174.955,38.442,157.347
C08619=1059.640,404.077,-118.213,174.962,38.450,157.350
C08620=1059.648,404.321,-118.257,174.969,38.458,157.352
C08621=1059.656,404.568,-118.300,174.976,38.466,157.354
C08622=1059.665,404.814,-118.343,174.983,38.474,157.356
C08623=1059.672,405.060,-118.387,174.990,38.483,157.358
C08624=1059.681,405.306,-118.430,174.996,38.491,157.361
C08625=1059.689,405.552,-118.474,175.002,38.500,157.363
C08626=1059.698,405.799,-118.518,175.009,38.508,157.365
C08627=1059.706,406.045,-118.561,175.016,38.516,157.367
C08628=1059.715,406.290,-118.605,175.023,38.525,157.370
C08629=1059.722,406.537,-118.649,175.030,38.534,157.372
C08630=1059.730,406.783,-118.693,175.037,38.542,157.374
C08631=1059.739,407.029,-118.736,175.044,38.550,157.377
C08632=1059.747,407.274,-118.780,175.051,38.559,157.379
C08633=1059.755,407.521,-118.824,175.058,38.567,157.381
C08634=1059.764,407.766,-118.868,175.065,38.576,157.384
C08635=1059.771,408.012,-118.911,175.072,38.585,157.386
C08636=1059.779,408.258,-118.956,175.079,38.593,157.388
C08637=1059.789,408.504,-119.000,175.086,38.602,157.391
C08638=1059.797,408.750,-119.044,175.093,38.610,157.393
C08639=1059.805,408.996,-119.088,175.100,38.619,157.395
C08640=1059.813,409.242,-119.132,175.107,38.628,157.398
C08641=1059.822,409.488,-119.176,175.116,38.637,157.400
C08642=1059.830,409.734,-119.221,175.123,38.646,157.402
C08643=1059.839,409.980,-119.264,175.130,38.655,157.405
C08644=1059.848,410.226,-119.309,175.137,38.663,157.407
C08645=1059.855,410.472,-119.353,175.144,38.672,157.410
C08646=1059.864,410.718,-119.396,175.151,38.681,157.412
C08647=1059.873,410.964,-119.442,175.158,38.690,157.414
C08648=1059.881,411.209,-119.486,175.166,38.699,157.417
C08649=1059.890,411.456,-119.531,175.174,38.708,157.419
C08650=1059.899,411.701,-119.575,175.181,38.716,157.422
C08651=1059.907,411.947,-119.619,175.188,38.725,157.424
C08652=1059.915,412.193,-119.664,175.195,38.734,157.427
C08653=1059.924,412.439,-119.707,175.203,38.743,157.429
C08654=1059.933,412.685,-119.753,175.210,38.753,157.432
C08655=1059.941,412.930,-119.797,175.218,38.762,157.434
C08656=1059.950,413.177,-119.842,175.225,38.770,157.437
C08657=1059.959,413.423,-119.887,175.233,38.780,157.439
C08658=1059.968,413.668,-119.931,175.240,38.789,157.442
C08659=1059.976,413.915,-119.976,175.248,38.798,157.444
C08660=1059.985,414.160,-120.021,175.256,38.807,157.447
C08661=1059.994,414.406,-120.065,175.263,38.816,157.449
C08662=1060.003,414.652,-120.111,175.270,38.826,157.452
C08663=1060.011,414.897,-120.156,175.279,38.835,157.454
C08664=1060.020,415.144,-120.201,175.286,38.845,157.457
C08665=1060.031,415.471,-120.261,175.296,38.857,157.460
C08666=1060.043,415.799,-120.322,175.306,38.870,157.464
C08667=1060.054,416.127,-120.382,175.317,38.882,157.467
C08668=1060.065,416.455,-120.442,175.328,38.895,157.471
C08669=1060.074,416.700,-120.487,175.335,38.904,157.473
C08670=1060.083,416.946,-120.533,175.343,38.914,157.476
C08671=1060.092,417.192,-120.578,175.351,38.923,157.479
C08672=1060.100,417.437,-120.623,175.359,38.932,157.481
C08673=1060.109,417.683,-120.669,175.367,38.942,157.484
C08674=1060.118,417.929,-120.714,175.375,38.952,157.487
C08675=1060.127,418.175,-120.760,175.383,38.962,157.490
C08676=1060.136,418.421,-120.805,175.391,38.971,157.492
C08677=1060.145,418.666,-120.850,175.398,38.981,157.495
C08678=1060.154,418.912,-120.897,175.407,38.991,157.498
C08679=1060.162,419.157,-120.942,175.415,39.000,157.500
C08680=1060.171,419.403,-120.988,175.423,39.010,157.503
C08681=1060.180,419.649,-121.033,175.432,39.020,157.506
C08682=1060.190,419.895,-121.080,175.439,39.030,157.509
C08683=1060.199,420.140,-121.125,175.448,39.040,157.511
C08684=1060.208,420.386,-121.172,175.456,39.050,157.514
C08685=1060.216,420.632,-121.217,175.464,39.060,157.517
C08686=1060.226,420.877,-121.263,175.472,39.069,157.520
C08687=1060.234,421.123,-121.309,175.481,39.080,157.523
C08688=1060.243,421.368,-121.355,175.489,39.090,157.525
C08689=1060.252,421.614,-121.402,175.497,39.100,157.528
C08690=1060.261,421.860,-121.448,175.506,39.110,157.531
C08691=1060.270,422.105,-121.494,175.515,39.120,157.534
C08692=1060.279,422.350,-121.540,175.522,39.130,157.537
C08693=1060.288,422.596,-121.587,175.531,39.140,157.540
C08694=1060.296,422.841,-121.633,175.540,39.150,157.543
C08695=1060.306,423.086,-121.679,175.548,39.161,157.546
C08696=1060.315,423.332,-121.727,175.556,39.171,157.548
C08697=1060.324,423.578,-121.773,175.565,39.181,157.551
C08698=1060.333,423.823,-121.819,175.573,39.192,157.554
C08699=1060.342,424.068,-121.866,175.582,39.202,157.557
C08700=1060.352,424.314,-121.912,175.591,39.212,157.560
C08701=1060.360,424.560,-121.959,175.600,39.222,157.563
C08702=1060.370,424.805,-122.005,175.609,39.233,157.566
C08703=1060.379,425.050,-122.052,175.617,39.243,157.569
C08704=1060.388,425.296,-122.099,175.626,39.254,157.572
C08705=1060.397,425.541,-122.146,175.634,39.265,157.575
C08706=1060.407,425.787,-122.193,175.643,39.275,157.578
C08707=1060.416,426.032,-122.240,175.652,39.286,157.581
C08708=1060.425,426.277,-122.286,175.661,39.296,157.584
C08709=1060.434,426.523,-122.333,175.670,39.307,157.587
C08710=1060.444,426.768,-122.380,175.679,39.318,157.590
C08711=1060.453,427.014,-122.427,175.688,39.329,157.594
C08712=1060.462,427.259,-122.475,175.698,39.339,157.597
C08713=1060.472,427.505,-122.521,175.707,39.350,157.600
C08714=1060.481,427.749,-122.569,175.715,39.361,157.603
C08715=1060.490,427.995,-122.617,175.724,39.372,157.606
C08716=1060.499,428.240,-122.664,175.734,39.383,157.609
C08717=1060.509,428.485,-122.711,175.743,39.394,157.612
C08718=1060.518,428.730,-122.759,175.752,39.404,157.615
C08719=1060.528,428.976,-122.807,175.761,39.415,157.619
C08720=1060.538,429.221,-122.854,175.771,39.427,157.622
C08721=1060.551,429.570,-122.921,175.783,39.442,157.626
C08722=1060.564,429.919,-122.989,175.797,39.458,157.631
C08723=1060.577,430.267,-123.057,175.810,39.474,157.636
C08724=1060.591,430.616,-123.125,175.824,39.490,157.640
C08725=1060.601,430.861,-123.172,175.833,39.501,157.644
C08726=1060.610,431.106,-123.221,175.843,39.512,157.647
C08727=1060.619,431.351,-123.268,175.852,39.524,157.650
C08728=1060.629,431.597,-123.316,175.861,39.535,157.654
C08729=1060.638,431.842,-123.365,175.872,39.546,157.657
C08730=1060.648,432.087,-123.413,175.881,39.558,157.660
C08731=1060.658,432.332,-123.461,175.890,39.570,157.664
C08732=1060.667,432.577,-123.509,175.901,39.581,157.667
C08733=1060.676,432.822,-123.557,175.910,39.592,157.670
C08734=1060.686,433.067,-123.606,175.920,39.604,157.674
C08735=1060.696,433.312,-123.654,175.930,39.616,157.677
C08736=1060.706,433.557,-123.703,175.940,39.627,157.681
C08737=1060.715,433.802,-123.751,175.949,39.639,157.684
C08738=1060.725,434.047,-123.800,175.960,39.651,157.688
C08739=1060.735,434.292,-123.848,175.969,39.662,157.691
C08740=1060.745,434.537,-123.897,175.980,39.674,157.695
C08741=1060.754,434.782,-123.945,175.989,39.686,157.698
C08742=1060.764,435.027,-123.994,176.000,39.698,157.702
C08743=1060.775,435.273,-124.043,176.009,39.710,157.705
C08744=1060.784,435.518,-124.091,176.020,39.722,157.709
C08745=1060.793,435.763,-124.140,176.030,39.733,157.712
C08746=1060.803,436.007,-124.190,176.040,39.745,157.716
C08747=1060.813,436.252,-124.238,176.050,39.758,157.719
C08748=1060.823,436.497,-124.287,176.061,39.770,157.723
C08749=1060.834,436.742,-124.336,176.071,39.782,157.727
C08750=1060.843,436.987,-124.385,176.081,39.794,157.730
C08751=1060.853,437.231,-124.434,176.092,39.806,157.734
C08752=1060.864,437.477,-124.483,176.103,39.818,157.738
C08753=1060.874,437.721,-124.532,176.113,39.830,157.741
C08754=1060.883,437.966,-124.582,176.123,39.843,157.745
C08755=1060.893,438.212,-124.631,176.134,39.855,157.749
C08756=1060.904,438.456,-124.680,176.145,39.868,157.752
C08757=1060.914,438.701,-124.730,176.156,39.880,157.756
C08758=1060.924,438.946,-124.779,176.166,39.893,157.760
C08759=1060.934,439.190,-124.829,176.177,39.905,157.764
C08760=1060.944,439.435,-124.878,176.188,39.918,157.768
C08761=1060.954,439.680,-124.928,176.199,39.930,157.771
C08762=1060.964,439.925,-124.978,176.210,39.943,157.775
C08763=1060.974,440.170,-125.028,176.221,39.956,157.779
C08764=1060.984,440.415,-125.077,176.232,39.968,157.783
C08765=1060.995,440.659,-125.128,176.243,39.981,157.787
C08766=1061.005,440.904,-125.177,176.254,39.993,157.791
C08767=1061.015,441.149,-125.227,176.265,40.006,157.795
C08768=1061.025,441.393,-125.278,176.276,40.019,157.798
C08769=1061.036,441.638,-125.327,176.287,40.032,157.802
C08770=1061.046,441.883,-125.378,176.298,40.045,157.806
C08771=1061.056,442.128,-125.428,176.309,40.058,157.810
C08772=1061.066,442.372,-125.478,176.321,40.071,157.814
C08773=1061.077,442.617,-125.528,176.332,40.085,157.818
C08774=1061.087,442.862,-125.579,176.343,40.098,157.822
C08775=1061.098,443.106,-125.629,176.354,40.110,157.826
C08776=1061.108,443.351,-125.680,176.367,40.124,157.831
C08777=1061.117,443.562,-125.723,176.376,40.135,157.834
C08778=1061.126,443.773,-125.767,176.386,40.147,157.838
C08779=1061.135,443.983,-125.811,176.397,40.158,157.841
C08780=1061.144,444.195,-125.854,176.407,40.170,157.845
C08781=1061.153,444.406,-125.899,176.416,40.181,157.848
C08782=1061.162,444.616,-125.942,176.427,40.193,157.852
C08783=1061.171,444.828,-125.986,176.437,40.205,157.855
C08784=1061.180,445.039,-126.030,176.447,40.216,157.859
C08785=1061.191,445.283,-126.080,176.459,40.230,157.863
C08786=1061.202,445.528,-126.132,176.470,40.244,157.868
C08787=1061.212,445.772,-126.183,176.483,40.257,157.872
C08788=1061.223,446.016,-126.234,176.495,40.271,157.876
C08789=1061.233,446.261,-126.285,176.507,40.284,157.880
C08790=1061.245,446.505,-126.336,176.519,40.298,157.885
C08791=1061.255,446.750,-126.387,176.531,40.312,157.889
C08792=1061.266,446.994,-126.439,176.544,40.326,157.893
C08793=1061.277,447.237,-126.489,176.556,40.340,157.898
C08794=1061.287,447.480,-126.540,176.568,40.353,157.902
C08795=1061.301,447.724,-126.590,176.580,40.367,157.906
C08796=1061.313,447.969,-126.640,176.593,40.380,157.910
C08797=1061.328,448.213,-126.689,176.605,40.393,157.915
C08798=1061.342,448.457,-126.737,176.619,40.406,157.919
C08799=1061.358,448.701,-126.785,176.631,40.418,157.923
C08800=1061.375,448.946,-126.832,176.644,40.430,157.927
C08801=1061.393,449.191,-126.879,176.656,40.443,157.931
C08802=1061.412,449.437,-126.925,176.669,40.454,157.934
C08803=1061.430,449.682,-126.970,176.682,40.466,157.938
C08804=1061.451,449.927,-127.015,176.695,40.477,157.942
C08805=1061.119,449.938,-127.290,176.690,40.593,157.974
C08806=1061.098,449.692,-127.246,176.677,40.582,157.970
C08807=1061.078,449.447,-127.200,176.664,40.570,157.966
C08808=1061.059,449.202,-127.155,176.651,40.559,157.962
C08809=1061.042,448.957,-127.109,176.637,40.547,157.958
C08810=1061.025,448.712,-127.061,176.624,40.534,157.954
C08811=1061.009,448.467,-127.013,176.612,40.522,157.950
C08812=1060.994,448.222,-126.965,176.598,40.509,157.946
C08813=1060.979,447.979,-126.916,176.586,40.497,157.942
C08814=1060.966,447.735,-126.866,176.573,40.483,157.938
C08815=1060.954,447.491,-126.817,176.561,40.470,157.934
C08816=1060.942,447.247,-126.766,176.548,40.457,157.929
C08817=1060.931,447.005,-126.715,176.537,40.443,157.925
C08818=1060.921,446.760,-126.663,176.524,40.429,157.921
C08819=1060.910,446.515,-126.612,176.511,40.415,157.916
C08820=1060.899,446.271,-126.561,176.500,40.401,157.912
C08821=1060.888,446.026,-126.510,176.487,40.388,157.908
C08822=1060.878,445.782,-126.458,176.476,40.374,157.903
C08823=1060.867,445.538,-126.408,176.463,40.361,157.899
C08824=1060.856,445.294,-126.356,176.452,40.347,157.895
C08825=1060.845,445.049,-126.306,176.439,40.333,157.891
C08826=1060.828,444.646,-126.221,176.420,40.311,157.884
C08827=1060.811,444.243,-126.138,176.400,40.289,157.877
C08828=1060.793,443.841,-126.054,176.380,40.267,157.870
C08829=1060.776,443.438,-125.971,176.361,40.245,157.863
C08830=1060.765,443.194,-125.920,176.350,40.232,157.859
C08831=1060.755,442.949,-125.870,176.339,40.219,157.855
C08832=1060.744,442.705,-125.819,176.326,40.206,157.851
C08833=1060.734,442.459,-125.769,176.315,40.193,157.847
C08834=1060.723,442.215,-125.719,176.304,40.180,157.843
C08835=1060.713,441.971,-125.668,176.293,40.167,157.839
C08836=1060.703,441.726,-125.619,176.282,40.154,157.835
C08837=1060.693,441.481,-125.568,176.270,40.141,157.831
C08838=1060.683,441.237,-125.518,176.258,40.128,157.827
C08839=1060.672,440.992,-125.467,176.247,40.115,157.823
C08840=1060.662,440.747,-125.418,176.236,40.103,157.819
C08841=1060.652,440.502,-125.368,176.225,40.090,157.815
C08842=1060.641,440.258,-125.318,176.214,40.077,157.812
C08843=1060.631,440.013,-125.268,176.203,40.065,157.808
C08844=1060.621,439.768,-125.218,176.192,40.052,157.804
C08845=1060.611,439.523,-125.169,176.181,40.040,157.800
C08846=1060.601,439.279,-125.119,176.170,40.027,157.796
C08847=1060.591,439.033,-125.069,176.160,40.015,157.792
C08848=1060.581,438.789,-125.020,176.149,40.002,157.789
C08849=1060.570,438.544,-124.970,176.138,39.990,157.785
C08850=1060.561,438.299,-124.921,176.127,39.978,157.781
C08851=1060.551,438.055,-124.871,176.116,39.965,157.777
C08852=1060.540,437.810,-124.822,176.105,39.953,157.774
C08853=1060.531,437.565,-124.773,176.096,39.940,157.770
C08854=1060.520,437.319,-124.723,176.085,39.928,157.766
C08855=1060.510,437.075,-124.674,176.074,39.916,157.763
C08856=1060.500,436.830,-124.625,176.063,39.904,157.759
C08857=1060.490,436.585,-124.576,176.054,39.892,157.755
C08858=1060.480,436.340,-124.527,176.043,39.880,157.752
C08859=1060.470,436.096,-124.478,176.032,39.868,157.748
C08860=1060.460,435.851,-124.429,176.022,39.856,157.745
C08861=1060.450,435.605,-124.380,176.012,39.844,157.741
C08862=1060.440,435.360,-124.332,176.002,39.833,157.737
C08863=1060.430,435.116,-124.283,175.991,39.820,157.734
C08864=1060.420,434.871,-124.234,175.982,39.809,157.730
C08865=1060.410,434.626,-124.186,175.971,39.797,157.727
C08866=1060.401,434.381,-124.137,175.961,39.785,157.723
C08867=1060.391,434.136,-124.088,175.951,39.774,157.720
C08868=1060.381,433.891,-124.040,175.940,39.762,157.716
C08869=1060.371,433.646,-123.991,175.931,39.750,157.713
C08870=1060.362,433.401,-123.943,175.920,39.738,157.709
C08871=1060.352,433.156,-123.894,175.911,39.727,157.706
C08872=1060.343,432.911,-123.845,175.901,39.715,157.703
C08873=1060.333,432.665,-123.797,175.891,39.704,157.699
C08874=1060.324,432.420,-123.749,175.882,39.692,157.696
C08875=1060.314,432.175,-123.700,175.872,39.681,157.692
C08876=1060.304,431.930,-123.653,175.862,39.669,157.689
C08877=1060.295,431.685,-123.604,175.852,39.658,157.686
C08878=1060.284,431.439,-123.557,175.843,39.646,157.682
C08879=1060.275,431.195,-123.509,175.833,39.635,157.679
C08880=1060.266,430.950,-123.461,175.823,39.624,157.676
C08881=1060.256,430.705,-123.412,175.814,39.613,157.672
C08882=1060.243,430.353,-123.344,175.800,39.597,157.668
C08883=1060.229,430.003,-123.275,175.787,39.581,157.663
C08884=1060.216,429.653,-123.208,175.773,39.565,157.658
C08885=1060.202,429.302,-123.139,175.760,39.549,157.654
C08886=1060.192,429.056,-123.092,175.750,39.538,157.650
C08887=1060.183,428.812,-123.044,175.741,39.528,157.647
C08888=1060.174,428.566,-122.996,175.732,39.516,157.644
C08889=1060.164,428.321,-122.949,175.723,39.506,157.641
C08890=1060.155,428.076,-122.902,175.713,39.494,157.638
C08891=1060.146,427.830,-122.855,175.704,39.484,157.635
C08892=1060.136,427.585,-122.808,175.695,39.473,157.631
C08893=1060.127,427.339,-122.760,175.686,39.462,157.628
C08894=1060.118,427.094,-122.712,175.677,39.451,157.625
C08895=1060.108,426.849,-122.666,175.668,39.441,157.622
C08896=1060.099,426.604,-122.618,175.659,39.430,157.619
C08897=1060.090,426.358,-122.571,175.650,39.419,157.616
C08898=1060.080,426.113,-122.525,175.641,39.409,157.613
C08899=1060.071,425.867,-122.477,175.632,39.398,157.610
C08900=1060.062,425.622,-122.431,175.623,39.387,157.607
C08901=1060.053,425.377,-122.384,175.614,39.377,157.604
C08902=1060.043,425.131,-122.337,175.605,39.367,157.601
C08903=1060.034,424.886,-122.290,175.596,39.356,157.598
C08904=1060.024,424.640,-122.243,175.588,39.346,157.595
C08905=1060.016,424.395,-122.196,175.579,39.336,157.592
C08906=1060.006,424.150,-122.150,175.570,39.325,157.589
C08907=1059.996,423.904,-122.103,175.561,39.315,157.586
C08908=1059.988,423.658,-122.057,175.553,39.304,157.583
C08909=1059.979,423.413,-122.010,175.544,39.294,157.580
C08910=1059.970,423.168,-121.964,175.536,39.284,157.577
C08911=1059.961,422.922,-121.918,175.527,39.274,157.574
C08912=1059.952,422.676,-121.870,175.518,39.264,157.571
C08913=1059.942,422.431,-121.824,175.509,39.253,157.568
C08914=1059.933,422.186,-121.778,175.502,39.244,157.566
C08915=1059.924,421.940,-121.731,175.493,39.233,157.563
C08916=1059.915,421.694,-121.686,175.484,39.223,157.560
C08917=1059.907,421.449,-121.639,175.476,39.213,157.557
C08918=1059.898,421.204,-121.593,175.468,39.203,157.554
C08919=1059.888,420.959,-121.547,175.459,39.193,157.551
C08920=1059.880,420.712,-121.501,175.451,39.183,157.548
C08921=1059.871,420.467,-121.455,175.443,39.173,157.546
C08922=1059.863,420.221,-121.409,175.434,39.163,157.543
C08923=1059.853,419.975,-121.362,175.426,39.153,157.540
C08924=1059.844,419.729,-121.317,175.418,39.143,157.537
C08925=1059.834,419.484,-121.271,175.410,39.134,157.534
C08926=1059.825,419.238,-121.225,175.401,39.124,157.532
C08927=1059.817,418.992,-121.180,175.394,39.115,157.529
C08928=1059.807,418.747,-121.134,175.385,39.105,157.526
C08929=1059.800,418.502,-121.088,175.377,39.095,157.523
C08930=1059.791,418.256,-121.043,175.369,39.086,157.521
C08931=1059.782,418.010,-120.997,175.361,39.076,157.518
C08932=1059.773,417.764,-120.952,175.353,39.066,157.515
C08933=1059.764,417.519,-120.907,175.345,39.056,157.513
C08934=1059.754,417.273,-120.860,175.337,39.047,157.510
C08935=1059.745,417.028,-120.815,175.330,39.038,157.507
C08936=1059.737,416.782,-120.770,175.321,39.028,157.505
C08937=1059.728,416.536,-120.725,175.314,39.019,157.502
C08938=1059.717,416.207,-120.664,175.302,39.006,157.499
C08939=1059.705,415.877,-120.603,175.292,38.993,157.495
C08940=1059.693,415.547,-120.542,175.282,38.981,157.491
C08941=1059.682,415.217,-120.482,175.272,38.968,157.488
C08942=1059.673,414.971,-120.436,175.263,38.959,157.485
C08943=1059.665,414.725,-120.392,175.256,38.949,157.483
C08944=1059.656,414.480,-120.346,175.248,38.941,157.480
C08945=1059.647,414.234,-120.301,175.240,38.931,157.478
C08946=1059.639,413.988,-120.257,175.233,38.922,157.475
C08947=1059.630,413.742,-120.211,175.225,38.913,157.473
C08948=1059.622,413.496,-120.167,175.217,38.903,157.470
C08949=1059.612,413.250,-120.123,175.210,38.895,157.468
C08950=1059.603,413.004,-120.077,175.203,38.886,157.465
C08951=1059.595,412.759,-120.033,175.195,38.876,157.463
C08952=1059.587,412.512,-119.988,175.187,38.867,157.460
C08953=1059.577,412.268,-119.944,175.180,38.859,157.458
C08954=1059.569,412.021,-119.899,175.172,38.850,157.455
C08955=1059.561,411.775,-119.855,175.165,38.841,157.453
C08956=1059.551,411.529,-119.811,175.158,38.832,157.450
C08957=1059.543,411.283,-119.766,175.150,38.823,157.448
C08958=1059.534,411.038,-119.721,175.143,38.814,157.445
C08959=1059.526,410.792,-119.677,175.135,38.805,157.443
C08960=1059.517,410.546,-119.633,175.128,38.796,157.441
C08961=1059.509,410.300,-119.588,175.121,38.787,157.438
C08962=1059.501,410.054,-119.544,175.114,38.778,157.436
C08963=1059.492,409.809,-119.500,175.106,38.770,157.433
C08964=1059.483,409.562,-119.456,175.099,38.761,157.431
C08965=1059.475,409.316,-119.412,175.092,38.752,157.429
C08966=1059.467,409.071,-119.368,175.084,38.744,157.426
C08967=1059.458,408.824,-119.323,175.077,38.735,157.424
C08968=1059.450,408.578,-119.279,175.070,38.726,157.421
C08969=1059.441,408.333,-119.235,175.063,38.718,157.419
C08970=1059.433,408.087,-119.192,175.056,38.709,157.417
C08971=1059.425,407.840,-119.147,175.049,38.701,157.414
C08972=1059.416,407.595,-119.103,175.042,38.692,157.412
C08973=1059.408,407.348,-119.060,175.035,38.683,157.410
C08974=1059.400,407.103,-119.015,175.028,38.675,157.407
C08975=1059.391,406.857,-118.972,175.021,38.666,157.405
C08976=1059.383,406.611,-118.928,175.014,38.658,157.403
C08977=1059.376,406.364,-118.884,175.007,38.650,157.401
C08978=1059.367,406.119,-118.841,175.000,38.641,157.398
C08979=1059.359,405.873,-118.797,174.993,38.633,157.396
C08980=1059.350,405.627,-118.753,174.986,38.624,157.394
C08981=1059.342,405.380,-118.709,174.979,38.616,157.391
C08982=1059.333,405.134,-118.666,174.972,38.607,157.389
C08983=1059.326,404.888,-118.623,174.966,38.599,157.387
C08984=1059.317,404.642,-118.579,174.959,38.591,157.385
C08985=1059.309,404.396,-118.535,174.952,38.583,157.383
C08986=1059.301,404.150,-118.492,174.945,38.575,157.380
C08987=1059.293,403.903,-118.449,174.938,38.566,157.378
C08988=1059.284,403.657,-118.405,174.931,38.558,157.376
C08989=1059.276,403.412,-118.363,174.924,38.550,157.374
C08990=1059.269,403.166,-118.319,174.917,38.542,157.372
C08991=1059.260,402.920,-118.276,174.911,38.533,157.369
C08992=1059.252,402.674,-118.233,174.904,38.525,157.367
C08993=1059.244,402.427,-118.190,174.898,38.518,157.365
C08994=1059.233,402.103,-118.132,174.889,38.507,157.362
C08995=1059.222,401.779,-118.076,174.880,38.496,157.359
C08996=1059.211,401.455,-118.020,174.871,38.486,157.357
C08997=1059.200,401.131,-117.963,174.863,38.475,157.354
C08998=1059.192,400.884,-117.921,174.856,38.467,157.352
C08999=1059.184,400.638,-117.877,174.849,38.459,157.349
C09000=1059.176,400.392,-117.834,174.843,38.451,157.347
C09001=1059.168,400.146,-117.792,174.837,38.444,157.345
C09002=1059.160,399.900,-117.749,174.830,38.436,157.343
C09003=1059.152,399.653,-117.707,174.823,38.428,157.341
C09004=1059.143,399.407,-117.664,174.816,38.420,157.339
C09005=1059.135,399.162,-117.621,174.811,38.412,157.337
C09006=1059.128,398.915,-117.578,174.804,38.404,157.335
C09007=1059.120,398.668,-117.536,174.797,38.397,157.333
C09008=1059.112,398.422,-117.493,174.791,38.389,157.331
C09009=1059.103,398.176,-117.451,174.785,38.381,157.329
C09010=1059.096,397.930,-117.408,174.778,38.374,157.327
C09011=1059.087,397.684,-117.366,174.772,38.366,157.325
C09012=1059.079,397.437,-117.323,174.766,38.358,157.323
C09013=1059.071,397.192,-117.281,174.759,38.350,157.321
C09014=1059.063,396.945,-117.238,174.753,38.343,157.319
C09015=1059.055,396.699,-117.197,174.747,38.335,157.317
C09016=1059.047,396.452,-117.154,174.740,38.328,157.315
C09017=1059.040,396.206,-117.112,174.734,38.320,157.313
C09018=1059.031,395.960,-117.070,174.728,38.313,157.311
C09019=1059.024,395.714,-117.027,174.722,38.305,157.309
C09020=1059.015,395.468,-116.985,174.715,38.297,157.307
C09021=1059.008,395.222,-116.943,174.709,38.290,157.305
C09022=1059.000,394.975,-116.901,174.703,38.282,157.303
C09023=1058.992,394.729,-116.859,174.696,38.275,157.301
C09024=1058.984,394.483,-116.817,174.691,38.267,157.299
C09025=1058.975,394.237,-116.775,174.684,38.261,157.297
C09026=1058.968,393.990,-116.734,174.679,38.253,157.295
C09027=1058.961,393.744,-116.692,174.672,38.246,157.293
C09028=1058.952,393.498,-116.650,174.665,38.238,157.291
C09029=1058.945,393.252,-116.608,174.660,38.231,157.289
C09030=1058.937,393.006,-116.566,174.653,38.224,157.287
C09031=1058.929,392.758,-116.524,174.648,38.216,157.285
C09032=1058.921,392.513,-116.483,174.641,38.209,157.284
C09033=1058.913,392.267,-116.441,174.635,38.202,157.282
C09034=1058.905,392.019,-116.399,174.629,38.195,157.280
C09035=1058.898,391.773,-116.357,174.623,38.187,157.278
C09036=1058.890,391.528,-116.316,174.617,38.180,157.276
C09037=1058.882,391.281,-116.275,174.611,38.173,157.274
C09038=1058.874,391.034,-116.232,174.605,38.166,157.272
C09039=1058.866,390.788,-116.192,174.599,38.158,157.270
C09040=1058.858,390.542,-116.150,174.594,38.151,157.268
C09041=1058.851,390.296,-116.109,174.587,38.144,157.267
C09042=1058.843,390.050,-116.067,174.582,38.137,157.265
C09043=1058.835,389.803,-116.026,174.575,38.130,157.263
C09044=1058.828,389.556,-115.984,174.570,38.123,157.261
C09045=1058.820,389.310,-115.944,174.563,38.116,157.259
C09046=1058.811,389.064,-115.902,174.558,38.109,157.257
C09047=1058.804,388.818,-115.861,174.552,38.102,157.256
C09048=1058.796,388.571,-115.821,174.546,38.095,157.254
C09049=1058.788,388.324,-115.779,174.540,38.088,157.252
C09050=1058.778,388.017,-115.728,174.533,38.079,157.250
C09051=1058.768,387.710,-115.677,174.526,38.071,157.248
C09052=1058.759,387.403,-115.626,174.518,38.062,157.245
C09053=1058.750,387.096,-115.574,174.511,38.054,157.243
C09054=1058.742,386.850,-115.534,174.506,38.047,157.241
C09055=1058.734,386.604,-115.493,174.499,38.040,157.240
C09056=1058.726,386.357,-115.452,174.494,38.033,157.238
C09057=1058.718,386.111,-115.411,174.489,38.026,157.236
C09058=1058.711,385.864,-115.370,174.482,38.019,157.234
C09059=1058.703,385.617,-115.330,174.477,38.013,157.233
C09060=1058.695,385.371,-115.289,174.471,38.006,157.231
C09061=1058.688,385.124,-115.248,174.465,37.999,157.229
